//     PlcTask Inputs/GVL_iXlinker.EtherCAT_Master_EMxxxx.Beckhoff_EM7xxx.A_0006_EM7004_0000_0018.ENC_Inputs_Channel_3.Latch_value <-> ENC Inputs Channel 3/Latch value
//     PlcTask Inputs/GVL_iXlinker.EtherCAT_Master_EMxxxx.Beckhoff_EM7xxx.A_0006_EM7004_0000_0018.ENC_Inputs_Channel_4.Latch_value <-> ENC Inputs Channel 4/Latch value
//     PlcTask Inputs/GVL_iXlinker.EtherCAT_Master_EMxxxx.Beckhoff_EM7xxx.A_0006_EM7004_0000_0018.PLS_Inputs.Status/PLS_Enabled <-> PLS Inputs/Status/PLS Enabled
//     PlcTask Inputs/GVL_iXlinker.EtherCAT_Master_EMxxxx.Beckhoff_EM7xxx.A_0006_EM7004_0000_0018.PLS_Inputs.Status/Unequal_SI_0 <-> PLS Inputs/Status/Unequal SI:0
//     PlcTask Outputs/GVL_iXlinker.EtherCAT_Master_EMxxxx.Beckhoff_EM7xxx.A_0006_EM7004_0000_0018.DO_Outputs.Output/Output_0 <-> DO Outputs/Output/Output 0
//     PlcTask Outputs/GVL_iXlinker.EtherCAT_Master_EMxxxx.Beckhoff_EM7xxx.A_0006_EM7004_0000_0018.DO_Outputs.Output/Output_1 <-> DO Outputs/Output/Output 1
//     PlcTask Outputs/GVL_iXlinker.EtherCAT_Master_EMxxxx.Beckhoff_EM7xxx.A_0006_EM7004_0000_0018.DO_Outputs.Output/Output_2 <-> DO Outputs/Output/Output 2
//     PlcTask Outputs/GVL_iXlinker.EtherCAT_Master_EMxxxx.Beckhoff_EM7xxx.A_0006_EM7004_0000_0018.DO_Outputs.Output/Output_3 <-> DO Outputs/Output/Output 3
//     PlcTask Outputs/GVL_iXlinker.EtherCAT_Master_EMxxxx.Beckhoff_EM7xxx.A_0006_EM7004_0000_0018.DO_Outputs.Output/Output_4 <-> DO Outputs/Output/Output 4
//     PlcTask Outputs/GVL_iXlinker.EtherCAT_Master_EMxxxx.Beckhoff_EM7xxx.A_0006_EM7004_0000_0018.DO_Outputs.Output/Output_5 <-> DO Outputs/Output/Output 5
//     PlcTask Outputs/GVL_iXlinker.EtherCAT_Master_EMxxxx.Beckhoff_EM7xxx.A_0006_EM7004_0000_0018.DO_Outputs.Output/Output_6 <-> DO Outputs/Output/Output 6
//     PlcTask Outputs/GVL_iXlinker.EtherCAT_Master_EMxxxx.Beckhoff_EM7xxx.A_0006_EM7004_0000_0018.DO_Outputs.Output/Output_7 <-> DO Outputs/Output/Output 7
//     PlcTask Outputs/GVL_iXlinker.EtherCAT_Master_EMxxxx.Beckhoff_EM7xxx.A_0006_EM7004_0000_0018.DO_Outputs.Output/Output_8 <-> DO Outputs/Output/Output 8
//     PlcTask Outputs/GVL_iXlinker.EtherCAT_Master_EMxxxx.Beckhoff_EM7xxx.A_0006_EM7004_0000_0018.DO_Outputs.Output/Output_9 <-> DO Outputs/Output/Output 9
//     PlcTask Outputs/GVL_iXlinker.EtherCAT_Master_EMxxxx.Beckhoff_EM7xxx.A_0006_EM7004_0000_0018.DO_Outputs.Output/Output_10 <-> DO Outputs/Output/Output 10
//     PlcTask Outputs/GVL_iXlinker.EtherCAT_Master_EMxxxx.Beckhoff_EM7xxx.A_0006_EM7004_0000_0018.DO_Outputs.Output/Output_11 <-> DO Outputs/Output/Output 11
//     PlcTask Outputs/GVL_iXlinker.EtherCAT_Master_EMxxxx.Beckhoff_EM7xxx.A_0006_EM7004_0000_0018.DO_Outputs.Output/Output_12 <-> DO Outputs/Output/Output 12
//     PlcTask Outputs/GVL_iXlinker.EtherCAT_Master_EMxxxx.Beckhoff_EM7xxx.A_0006_EM7004_0000_0018.DO_Outputs.Output/Output_13 <-> DO Outputs/Output/Output 13
//     PlcTask Outputs/GVL_iXlinker.EtherCAT_Master_EMxxxx.Beckhoff_EM7xxx.A_0006_EM7004_0000_0018.DO_Outputs.Output/Output_14 <-> DO Outputs/Output/Output 14
//     PlcTask Outputs/GVL_iXlinker.EtherCAT_Master_EMxxxx.Beckhoff_EM7xxx.A_0006_EM7004_0000_0018.DO_Outputs.Output/Output_15 <-> DO Outputs/Output/Output 15
//     PlcTask Outputs/GVL_iXlinker.EtherCAT_Master_EMxxxx.Beckhoff_EM7xxx.A_0006_EM7004_0000_0018.AO_Outputs_Channel_1.Analog_output <-> AO Outputs Channel 1/Analog output
//     PlcTask Outputs/GVL_iXlinker.EtherCAT_Master_EMxxxx.Beckhoff_EM7xxx.A_0006_EM7004_0000_0018.AO_Outputs_Channel_2.Analog_output <-> AO Outputs Channel 2/Analog output
//     PlcTask Outputs/GVL_iXlinker.EtherCAT_Master_EMxxxx.Beckhoff_EM7xxx.A_0006_EM7004_0000_0018.AO_Outputs_Channel_3.Analog_output <-> AO Outputs Channel 3/Analog output
//     PlcTask Outputs/GVL_iXlinker.EtherCAT_Master_EMxxxx.Beckhoff_EM7xxx.A_0006_EM7004_0000_0018.AO_Outputs_Channel_4.Analog_output <-> AO Outputs Channel 4/Analog output
//     PlcTask Outputs/GVL_iXlinker.EtherCAT_Master_EMxxxx.Beckhoff_EM7xxx.A_0006_EM7004_0000_0018.ENC_Outputs_Channel_1.Control/Enable_latch_extern_on_positive_edge <-> ENC Outputs Channel 1/Control/Enable latch extern on positive edge
//     PlcTask Outputs/GVL_iXlinker.EtherCAT_Master_EMxxxx.Beckhoff_EM7xxx.A_0006_EM7004_0000_0018.ENC_Outputs_Channel_2.Control/Enable_latch_extern_on_positive_edge <-> ENC Outputs Channel 2/Control/Enable latch extern on positive edge
//     PlcTask Outputs/GVL_iXlinker.EtherCAT_Master_EMxxxx.Beckhoff_EM7xxx.A_0006_EM7004_0000_0018.ENC_Outputs_Channel_3.Control/Enable_latch_extern_on_positive_edge <-> ENC Outputs Channel 3/Control/Enable latch extern on positive edge
//     PlcTask Outputs/GVL_iXlinker.EtherCAT_Master_EMxxxx.Beckhoff_EM7xxx.A_0006_EM7004_0000_0018.ENC_Outputs_Channel_4.Control/Enable_latch_extern_on_positive_edge <-> ENC Outputs Channel 4/Control/Enable latch extern on positive edge
//     PlcTask Outputs/GVL_iXlinker.EtherCAT_Master_EMxxxx.Beckhoff_EM7xxx.A_0006_EM7004_0000_0018.ENC_Outputs_Channel_1.Control/Set_counter <-> ENC Outputs Channel 1/Control/Set counter
//     PlcTask Outputs/GVL_iXlinker.EtherCAT_Master_EMxxxx.Beckhoff_EM7xxx.A_0006_EM7004_0000_0018.ENC_Outputs_Channel_2.Control/Set_counter <-> ENC Outputs Channel 2/Control/Set counter
//     PlcTask Outputs/GVL_iXlinker.EtherCAT_Master_EMxxxx.Beckhoff_EM7xxx.A_0006_EM7004_0000_0018.ENC_Outputs_Channel_3.Control/Set_counter <-> ENC Outputs Channel 3/Control/Set counter
//     PlcTask Outputs/GVL_iXlinker.EtherCAT_Master_EMxxxx.Beckhoff_EM7xxx.A_0006_EM7004_0000_0018.ENC_Outputs_Channel_4.Control/Set_counter <-> ENC Outputs Channel 4/Control/Set counter
//     PlcTask Outputs/GVL_iXlinker.EtherCAT_Master_EMxxxx.Beckhoff_EM7xxx.A_0006_EM7004_0000_0018.ENC_Outputs_Channel_1.Control/Enable_latch_extern_on_negative_edge <-> ENC Outputs Channel 1/Control/Enable latch extern on negative edge
//     PlcTask Outputs/GVL_iXlinker.EtherCAT_Master_EMxxxx.Beckhoff_EM7xxx.A_0006_EM7004_0000_0018.ENC_Outputs_Channel_2.Control/Enable_latch_extern_on_negative_edge <-> ENC Outputs Channel 2/Control/Enable latch extern on negative edge
//     PlcTask Outputs/GVL_iXlinker.EtherCAT_Master_EMxxxx.Beckhoff_EM7xxx.A_0006_EM7004_0000_0018.ENC_Outputs_Channel_3.Control/Enable_latch_extern_on_negative_edge <-> ENC Outputs Channel 3/Control/Enable latch extern on negative edge
//     PlcTask Outputs/GVL_iXlinker.EtherCAT_Master_EMxxxx.Beckhoff_EM7xxx.A_0006_EM7004_0000_0018.ENC_Outputs_Channel_4.Control/Enable_latch_extern_on_negative_edge <-> ENC Outputs Channel 4/Control/Enable latch extern on negative edge
//     PlcTask Outputs/GVL_iXlinker.EtherCAT_Master_EMxxxx.Beckhoff_EM7xxx.A_0006_EM7004_0000_0018.ENC_Outputs_Channel_1.Set_counter_value <-> ENC Outputs Channel 1/Set counter value
//     PlcTask Outputs/GVL_iXlinker.EtherCAT_Master_EMxxxx.Beckhoff_EM7xxx.A_0006_EM7004_0000_0018.ENC_Outputs_Channel_2.Set_counter_value <-> ENC Outputs Channel 2/Set counter value
//     PlcTask Outputs/GVL_iXlinker.EtherCAT_Master_EMxxxx.Beckhoff_EM7xxx.A_0006_EM7004_0000_0018.ENC_Outputs_Channel_3.Set_counter_value <-> ENC Outputs Channel 3/Set counter value
//     PlcTask Outputs/GVL_iXlinker.EtherCAT_Master_EMxxxx.Beckhoff_EM7xxx.A_0006_EM7004_0000_0018.ENC_Outputs_Channel_4.Set_counter_value <-> ENC Outputs Channel 4/Set counter value
//     PlcTask Outputs/GVL_iXlinker.EtherCAT_Master_EMxxxx.Beckhoff_EM7xxx.A_0006_EM7004_0000_0018.PLS_Outputs.Control/Enable_PLS <-> PLS Outputs/Control/Enable PLS
//     PlcTask Inputs/GVL_iXlinker.EtherCAT_Master_EMxxxx.Beckhoff_EM7xxx.A_0006_EM7004_0000_0018.WcState.WcState <-> WcState/WcState
//     PlcTask Inputs/GVL_iXlinker.EtherCAT_Master_EMxxxx.Beckhoff_EM7xxx.A_0006_EM7004_0000_0018.WcState.InputToggle <-> WcState/InputToggle
//     PlcTask Inputs/GVL_iXlinker.EtherCAT_Master_EMxxxx.Beckhoff_EM7xxx.A_0006_EM7004_0000_0018.InfoData.AdsAddr <-> InfoData/AdsAddr
//     PlcTask Inputs/GVL_iXlinker.EtherCAT_Master_EMxxxx.Beckhoff_EM7xxx.A_0006_EM7004_0000_0018.InfoData.State <-> InfoData/State
//   PLC/PLC Instance <-> EtherCAT_Master_EMxxxx
//     PlcTask Inputs/GVL_iXlinker.EtherCAT_Master_EMxxxx.SyncUnits._default._unreferenced.WcState.WcState <-> SyncUnits/<default>/<unreferenced>/WcState/WcState
//     PlcTask Inputs/GVL_iXlinker.EtherCAT_Master_EMxxxx.SyncUnits._default._unreferenced.InfoData.ObjectId <-> SyncUnits/<default>/<unreferenced>/InfoData/ObjectId
//     PlcTask Inputs/GVL_iXlinker.EtherCAT_Master_EMxxxx.SyncUnits._default._unreferenced.InfoData.State <-> SyncUnits/<default>/<unreferenced>/InfoData/State
//     PlcTask Inputs/GVL_iXlinker.EtherCAT_Master_EMxxxx.SyncUnits._default._unreferenced.InfoData.SlaveCount <-> SyncUnits/<default>/<unreferenced>/InfoData/SlaveCount
//     PlcTask Inputs/GVL_iXlinker.EtherCAT_Master_EMxxxx.SyncUnits._default.PlcTask.WcState.WcState <-> SyncUnits/<default>/PlcTask/WcState/WcState
//     PlcTask Inputs/GVL_iXlinker.EtherCAT_Master_EMxxxx.SyncUnits._default.PlcTask.InfoData.ObjectId <-> SyncUnits/<default>/PlcTask/InfoData/ObjectId
//     PlcTask Inputs/GVL_iXlinker.EtherCAT_Master_EMxxxx.SyncUnits._default.PlcTask.InfoData.State <-> SyncUnits/<default>/PlcTask/InfoData/State
//     PlcTask Inputs/GVL_iXlinker.EtherCAT_Master_EMxxxx.SyncUnits._default.PlcTask.InfoData.SlaveCount <-> SyncUnits/<default>/PlcTask/InfoData/SlaveCount
//     PlcTask Inputs/GVL_iXlinker.EtherCAT_Master_EMxxxx.Inputs.SlaveCount <-> Inputs/SlaveCount
//     PlcTask Inputs/GVL_iXlinker.EtherCAT_Master_EMxxxx.Inputs.DevState <-> Inputs/DevState
//     PlcTask Inputs/GVL_iXlinker.EtherCAT_Master_EMxxxx.Inputs.Frm{0..25}State <-> Inputs/Frm{0..25}State  (26 links)
//     PlcTask Inputs/GVL_iXlinker.EtherCAT_Master_EMxxxx.Inputs.Frm{0..25}WcState <-> Inputs/Frm{0..25}WcState  (26 links)
//     PlcTask Inputs/GVL_iXlinker.EtherCAT_Master_EMxxxx.Inputs.Frm{0..25}InputToggle <-> Inputs/Frm{0..25}InputToggle  (26 links)
//     PlcTask Outputs/GVL_iXlinker.EtherCAT_Master_EMxxxx.Outputs.DevCtrl <-> Outputs/DevCtrl
//     PlcTask Outputs/GVL_iXlinker.EtherCAT_Master_EMxxxx.Outputs.Frm{0..25}Ctrl <-> Outputs/Frm{0..25}Ctrl  (26 links)
//     PlcTask Outputs/GVL_iXlinker.EtherCAT_Master_EMxxxx.Outputs.Frm{0..25}WcCtrl <-> Outputs/Frm{0..25}WcCtrl  (26 links)
//     PlcTask Inputs/GVL_iXlinker.EtherCAT_Master_EMxxxx.InfoData.ChangeCount <-> InfoData/ChangeCount
//     PlcTask Inputs/GVL_iXlinker.EtherCAT_Master_EMxxxx.InfoData.DevId <-> InfoData/DevId
//     PlcTask Inputs/GVL_iXlinker.EtherCAT_Master_EMxxxx.InfoData.AmsNetId <-> InfoData/AmsNetId
//     PlcTask Inputs/GVL_iXlinker.EtherCAT_Master_EMxxxx.InfoData.CfgSlaveCount <-> InfoData/CfgSlaveCount
//     PlcTask Inputs/GVL_iXlinker.EtherCAT_Master_EMxxxx.InfoData.DcToTcTimeOffset <-> InfoData/DcToTcTimeOffset
//     PlcTask Inputs/GVL_iXlinker.EtherCAT_Master_EMxxxx.InfoData.DcToExtTimeOffset <-> InfoData/DcToExtTimeOffset

CONFIGURATION PLC
    RESOURCE PLC ON TwinCAT3
        TASK PlcTask(INTERVAL := T#10ms, PRIORITY := 20);
        PROGRAM MAIN WITH PlcTask : MAIN;
    END_RESOURCE
END_CONFIGURATION

// ---- DUTs/IO/PdoEntries/Status_E3F6A94B.TcDUT
{attribute 'GeneratedUsingTerminal: EM3701-0000-0016'}
{attribute addProperty BoxType "EM3701-0000-0016"}
{attribute addProperty Id "UnderrangeBOOL1OverrangeBOOL1Limit_1BYTE1Limit_2BYTE1ErrorBOOL1TxPDO_StateBOOL1"}
{attribute addProperty CRC "3824593227"}
{attribute addProperty Size "6"}
TYPE Status_E3F6A94B :
STRUCT
	{attribute addProperty Name "Underrange"}
	Underrange : BOOL;
	{attribute addProperty Name "Overrange"}
	Overrange : BOOL;
	{attribute addProperty Name "Limit_1"}
	Limit_1 : BYTE;
	{attribute addProperty Name "Limit_2"}
	Limit_2 : BYTE;
	{attribute addProperty Name "Error"}
	Error : BOOL;
	{attribute addProperty Name "TxPDO_State"}
	TxPDO_State : BOOL;
END_STRUCT
END_TYPE

// ---- DUTs/IO/PdoEntries/Input_97D1F313.TcDUT
{attribute 'GeneratedUsingTerminal: EM7004-0000-0017'}
{attribute addProperty BoxType "EM7004-0000-0017"}
{attribute addProperty Id "Input_0BOOL1Input_1BOOL1Input_2BOOL1Input_3BOOL1Input_4BOOL1Input_5BOOL1Input_6BOOL1Input_7BOOL1Input_8BOOL1Input_9BOOL1Input_10BOOL1Input_11BOOL1Input_12BOOL1Input_13BOOL1Input_14BOOL1Input_15BOOL1"}
{attribute addProperty CRC "2547118867"}
{attribute addProperty Size "16"}
TYPE Input_97D1F313 :
STRUCT
	{attribute addProperty Name "Input_0"}
	Input_0 : BOOL;
	{attribute addProperty Name "Input_1"}
	Input_1 : BOOL;
	{attribute addProperty Name "Input_2"}
	Input_2 : BOOL;
	{attribute addProperty Name "Input_3"}
	Input_3 : BOOL;
	{attribute addProperty Name "Input_4"}
	Input_4 : BOOL;
	{attribute addProperty Name "Input_5"}
	Input_5 : BOOL;
	{attribute addProperty Name "Input_6"}
	Input_6 : BOOL;
	{attribute addProperty Name "Input_7"}
	Input_7 : BOOL;
	{attribute addProperty Name "Input_8"}
	Input_8 : BOOL;
	{attribute addProperty Name "Input_9"}
	Input_9 : BOOL;
	{attribute addProperty Name "Input_10"}
	Input_10 : BOOL;
	{attribute addProperty Name "Input_11"}
	Input_11 : BOOL;
	{attribute addProperty Name "Input_12"}
	Input_12 : BOOL;
	{attribute addProperty Name "Input_13"}
	Input_13 : BOOL;
	{attribute addProperty Name "Input_14"}
	Input_14 : BOOL;
	{attribute addProperty Name "Input_15"}
	Input_15 : BOOL;
END_STRUCT
END_TYPE

// ---- DUTs/IO/PdoEntries/Status_B4798D86.TcDUT
{attribute 'GeneratedUsingTerminal: EM7004-0000-0017'}
{attribute addProperty BoxType "EM7004-0000-0017"}
{attribute addProperty Id "Latch_extern_validBOOL1Set_counter_doneBOOL1Status_of_input_ABOOL1Status_of_input_BBOOL1Status_of_input_gateBOOL1Status_of_extern_latchBOOL1TxPDO_ToggleBOOL1"}
{attribute addProperty CRC "3027864966"}
{attribute addProperty Size "7"}
TYPE Status_B4798D86 :
STRUCT
	{attribute addProperty Name "Latch_extern_valid"}
	Latch_extern_valid : BOOL;
	{attribute addProperty Name "Set_counter_done"}
	Set_counter_done : BOOL;
	{attribute addProperty Name "Status_of_input_A"}
	Status_of_input_A : BOOL;
	{attribute addProperty Name "Status_of_input_B"}
	Status_of_input_B : BOOL;
	{attribute addProperty Name "Status_of_input_gate"}
	Status_of_input_gate : BOOL;
	{attribute addProperty Name "Status_of_extern_latch"}
	Status_of_extern_latch : BOOL;
	{attribute addProperty Name "TxPDO_Toggle"}
	TxPDO_Toggle : BOOL;
END_STRUCT
END_TYPE

// ---- DUTs/IO/PdoEntries/Status_882A150F.TcDUT
{attribute 'GeneratedUsingTerminal: EM7004-0000-0017'}
{attribute addProperty BoxType "EM7004-0000-0017"}
{attribute addProperty Id "PLS_EnabledBOOL1Unequal_SI_0BOOL1"}
{attribute addProperty CRC "2284459279"}
{attribute addProperty Size "2"}
TYPE Status_882A150F :
STRUCT
	{attribute addProperty Name "PLS_Enabled"}
	PLS_Enabled : BOOL;
	{attribute addProperty Name "Unequal_SI_0"}
	Unequal_SI_0 : BOOL;
END_STRUCT
END_TYPE

// ---- DUTs/IO/PdoEntries/Output_FFFF807A.TcDUT
{attribute 'GeneratedUsingTerminal: EM7004-0000-0017'}
{attribute addProperty BoxType "EM7004-0000-0017"}
{attribute addProperty Id "Output_0BOOL1Output_1BOOL1Output_2BOOL1Output_3BOOL1Output_4BOOL1Output_5BOOL1Output_6BOOL1Output_7BOOL1Output_8BOOL1Output_9BOOL1Output_10BOOL1Output_11BOOL1Output_12BOOL1Output_13BOOL1Output_14BOOL1Output_15BOOL1"}
{attribute addProperty CRC "4294934650"}
{attribute addProperty Size "16"}
TYPE Output_FFFF807A :
STRUCT
	{attribute addProperty Name "Output_0"}
	Output_0 : BOOL;
	{attribute addProperty Name "Output_1"}
	Output_1 : BOOL;
	{attribute addProperty Name "Output_2"}
	Output_2 : BOOL;
	{attribute addProperty Name "Output_3"}
	Output_3 : BOOL;
	{attribute addProperty Name "Output_4"}
	Output_4 : BOOL;
	{attribute addProperty Name "Output_5"}
	Output_5 : BOOL;
	{attribute addProperty Name "Output_6"}
	Output_6 : BOOL;
	{attribute addProperty Name "Output_7"}
	Output_7 : BOOL;
	{attribute addProperty Name "Output_8"}
	Output_8 : BOOL;
	{attribute addProperty Name "Output_9"}
	Output_9 : BOOL;
	{attribute addProperty Name "Output_10"}
	Output_10 : BOOL;
	{attribute addProperty Name "Output_11"}
	Output_11 : BOOL;
	{attribute addProperty Name "Output_12"}
	Output_12 : BOOL;
	{attribute addProperty Name "Output_13"}
	Output_13 : BOOL;
	{attribute addProperty Name "Output_14"}
	Output_14 : BOOL;
	{attribute addProperty Name "Output_15"}
	Output_15 : BOOL;
END_STRUCT
END_TYPE

// ---- DUTs/IO/PdoEntries/Control_F189B737.TcDUT
{attribute 'GeneratedUsingTerminal: EM7004-0000-0017'}
{attribute addProperty BoxType "EM7004-0000-0017"}
{attribute addProperty Id "Enable_latch_extern_on_positive_edgeBOOL1Set_counterBOOL1Enable_latch_extern_on_negative_edgeBOOL1"}
{attribute addProperty CRC "4052334391"}
{attribute addProperty Size "3"}
TYPE Control_F189B737 :
STRUCT
	{attribute addProperty Name "Enable_latch_extern_on_positive_edge"}
	Enable_latch_extern_on_positive_edge : BOOL;
	{attribute addProperty Name "Set_counter"}
	Set_counter : BOOL;
	{attribute addProperty Name "Enable_latch_extern_on_negative_edge"}
	Enable_latch_extern_on_negative_edge : BOOL;
END_STRUCT
END_TYPE

// ---- DUTs/IO/PdoEntries/Control_17BA1FC2.TcDUT
{attribute 'GeneratedUsingTerminal: EM7004-0000-0017'}
{attribute addProperty BoxType "EM7004-0000-0017"}
{attribute addProperty Id "Enable_PLSBOOL1"}
{attribute addProperty CRC "398073794"}
{attribute addProperty Size "1"}
TYPE Control_17BA1FC2 :
STRUCT
	{attribute addProperty Name "Enable_PLS"}
	Enable_PLS : BOOL;
END_STRUCT
END_TYPE

// ---- DUTs/IO/PDOs/InfoData_6F19DB2B.TcDUT
{attribute 'GeneratedUsingTerminal: EK1100-0000-0018'}
{attribute addProperty BoxType "EK1100-0000-0018"}
{attribute addProperty Id "StateAT %I*UINT2"}
{attribute addProperty CRC "1863965483"}
{attribute addProperty Size "2"}
TYPE InfoData_6F19DB2B :
STRUCT
	{attribute addProperty Name "State"}
	State AT %I* : UINT;
END_STRUCT
END_TYPE

// ---- DUTs/IO/PDOs/Channel_42CA91F7.TcDUT
{attribute 'GeneratedUsingTerminal: EM2042-0000-0016'}
{attribute addProperty BoxType "EM2042-0000-0016"}
{attribute addProperty Id "OutputAT %Q*BOOL1"}
{attribute addProperty CRC "1120571895"}
{attribute addProperty Size "1"}
TYPE Channel_42CA91F7 EXTENDS OutputBase_10CEE7DE :
STRUCT
	{attribute addProperty Name "Output"}
	Output AT %Q* : BOOL;
END_STRUCT
END_TYPE

// ---- DUTs/IO/PDOs/WcState_0B2B16F9.TcDUT
{attribute 'GeneratedUsingTerminal: EM2042-0000-0016'}
{attribute addProperty BoxType "EM2042-0000-0016"}
{attribute addProperty Id "WcStateAT %I*BOOL1"}
{attribute addProperty CRC "187373305"}
{attribute addProperty Size "1"}
TYPE WcState_0B2B16F9 :
STRUCT
	{attribute addProperty Name "WcState"}
	WcState AT %I* : BOOL;
END_STRUCT
END_TYPE

// ---- DUTs/IO/PDOs/AI_Inputs_5AF6604E.TcDUT
{attribute 'GeneratedUsingTerminal: EM3701-0000-0016'}
{attribute addProperty BoxType "EM3701-0000-0016"}
{attribute addProperty Id "StatusAT %I*Status_E3F6A94B6ValueAT %I*INT2"}
{attribute addProperty CRC "1526095950"}
{attribute addProperty Size "8"}
TYPE AI_Inputs_5AF6604E EXTENDS InputBase_8311D824 :
STRUCT
	{attribute addProperty Name "Status"}
	Status AT %I* : Status_E3F6A94B;
	{attribute addProperty Name "Value"}
	Value AT %I* : INT;
END_STRUCT
END_TYPE

// ---- DUTs/IO/PDOs/WcState_9091E0EB.TcDUT
{attribute 'GeneratedUsingTerminal: EM3701-0000-0016'}
{attribute addProperty BoxType "EM3701-0000-0016"}
{attribute addProperty Id "WcStateAT %I*BOOL1InputToggleAT %I*BOOL1"}
{attribute addProperty CRC "2425479403"}
{attribute addProperty Size "2"}
TYPE WcState_9091E0EB :
STRUCT
	{attribute addProperty Name "WcState"}
	WcState AT %I* : BOOL;
	{attribute addProperty Name "InputToggle"}
	InputToggle AT %I* : BOOL;
END_STRUCT
END_TYPE

// ---- DUTs/IO/PDOs/InfoData_32EB74EA.TcDUT
{attribute 'GeneratedUsingTerminal: EM3701-0000-0016'}
{attribute addProperty BoxType "EM3701-0000-0016"}
{attribute addProperty Id "AdsAddrAT %I*AMSADDR8StateAT %I*UINT2"}
{attribute addProperty CRC "854291690"}
{attribute addProperty Size "10"}
TYPE InfoData_32EB74EA EXTENDS InputBase_8311D824 :
STRUCT
	{attribute addProperty Name "AdsAddr"}
	AdsAddr AT %I* : AMSADDR;
	{attribute addProperty Name "State"}
	State AT %I* : UINT;
END_STRUCT
END_TYPE

// ---- DUTs/IO/PDOs/AI_Input_Channel_5AF6604E.TcDUT
{attribute 'GeneratedUsingTerminal: EM3702-0000-0016'}
{attribute addProperty BoxType "EM3702-0000-0016"}
{attribute addProperty Id "StatusAT %I*Status_E3F6A94B6ValueAT %I*INT2"}
{attribute addProperty CRC "1526095950"}
{attribute addProperty Size "8"}
TYPE AI_Input_Channel_5AF6604E EXTENDS InputBase_8311D824 :
STRUCT
	{attribute addProperty Name "Status"}
	Status AT %I* : Status_E3F6A94B;
	{attribute addProperty Name "Value"}
	Value AT %I* : INT;
END_STRUCT
END_TYPE

// ---- DUTs/IO/PDOs/Digital_BD004D6F.TcDUT
{attribute 'GeneratedUsingTerminal: EM7004-0000-9995'}
{attribute addProperty BoxType "EM7004-0000-9995"}
{attribute addProperty Id "InputAT %I*ARRAY[0..15] OF BOOL16"}
{attribute addProperty CRC "2621435360"}
{attribute addProperty Size "16"}
TYPE Digital_BD004D6F EXTENDS InputBase_8311D824 :
STRUCT
	{attribute addProperty Name "Input"}
	Input AT %I* : ARRAY[0..15] OF BOOL;
END_STRUCT
END_TYPE

// ---- DUTs/IO/PDOs/Encoder_Channel_2E4EA213.TcDUT
{attribute 'GeneratedUsingTerminal: EM7004-0000-9995'}
{attribute addProperty BoxType "EM7004-0000-9995"}
{attribute addProperty Id "StatusAT %I*UINT2ValueAT %I*UINT2LatchAT %I*UINT2"}
{attribute addProperty CRC "776905235"}
{attribute addProperty Size "6"}
TYPE Encoder_Channel_2E4EA213 EXTENDS InputBase_8311D824 :
STRUCT
	{attribute addProperty Name "Status"}
	Status AT %I* : UINT;
	{attribute addProperty Name "Value"}
	Value AT %I* : UINT;
	{attribute addProperty Name "Latch"}
	Latch AT %I* : UINT;
END_STRUCT
END_TYPE

// ---- DUTs/IO/PDOs/Digital_A7E1DFAB.TcDUT
{attribute 'GeneratedUsingTerminal: EM7004-0000-9995'}
{attribute addProperty BoxType "EM7004-0000-9995"}
{attribute addProperty Id "OutputAT %Q*ARRAY[0..15] OF BOOL16"}
{attribute addProperty CRC "1538723034"}
{attribute addProperty Size "16"}
TYPE Digital_A7E1DFAB EXTENDS OutputBase_10CEE7DE :
STRUCT
	{attribute addProperty Name "Output"}
	Output AT %Q* : ARRAY[0..15] OF BOOL;
END_STRUCT
END_TYPE

// ---- DUTs/IO/PDOs/Analog_Channel_5F9B7EA6.TcDUT
{attribute 'GeneratedUsingTerminal: EM7004-0000-9995'}
{attribute addProperty BoxType "EM7004-0000-9995"}
{attribute addProperty Id "OutputAT %Q*INT2"}
{attribute addProperty CRC "1604026022"}
{attribute addProperty Size "2"}
TYPE Analog_Channel_5F9B7EA6 EXTENDS OutputBase_10CEE7DE :
STRUCT
	{attribute addProperty Name "Output"}
	Output AT %Q* : INT;
END_STRUCT
END_TYPE

// ---- DUTs/IO/PDOs/Encoder_Channel_B7999E14.TcDUT
{attribute 'GeneratedUsingTerminal: EM7004-0000-9995'}
{attribute addProperty BoxType "EM7004-0000-9995"}
{attribute addProperty Id "CtrlAT %Q*UINT2ValueAT %Q*UINT2"}
{attribute addProperty CRC "3080298004"}
{attribute addProperty Size "4"}
TYPE Encoder_Channel_B7999E14 EXTENDS OutputBase_10CEE7DE :
STRUCT
	{attribute addProperty Name "Ctrl"}
	Ctrl AT %Q* : UINT;
	{attribute addProperty Name "Value"}
	Value AT %Q* : UINT;
END_STRUCT
END_TYPE

// ---- DUTs/IO/PDOs/DI_Inputs_BD004D6F.TcDUT
{attribute 'GeneratedUsingTerminal: EM7004-0000-9996'}
{attribute addProperty BoxType "EM7004-0000-9996"}
{attribute addProperty Id "InputAT %I*ARRAY[0..15] OF BOOL16"}
{attribute addProperty CRC "2621435360"}
{attribute addProperty Size "16"}
TYPE DI_Inputs_BD004D6F EXTENDS InputBase_8311D824 :
STRUCT
	{attribute addProperty Name "Input"}
	Input AT %I* : ARRAY[0..15] OF BOOL;
END_STRUCT
END_TYPE

// ---- DUTs/IO/PDOs/ENC_Inputs_Channel_69C51E8E.TcDUT
{attribute 'GeneratedUsingTerminal: EM7004-0000-9996'}
{attribute addProperty BoxType "EM7004-0000-9996"}
{attribute addProperty Id "Latch_extern_validAT %I*BOOL1Set_counter_doneAT %I*BOOL1Status_of_input_AAT %I*BOOL1Status_of_input_BAT %I*BOOL1Status_of_input_gateAT %I*BOOL1Status_of_extern_latchAT %I*BOOL1Counter_valueAT %I*UINT2Latch_valueAT %I*UINT2"}
{attribute addProperty CRC "1774526094"}
{attribute addProperty Size "10"}
TYPE ENC_Inputs_Channel_69C51E8E EXTENDS InputBase_8311D824 :
STRUCT
	{attribute addProperty Name "Latch_extern_valid"}
	Latch_extern_valid AT %I* : BOOL;
	{attribute addProperty Name "Set_counter_done"}
	Set_counter_done AT %I* : BOOL;
	{attribute addProperty Name "Status_of_input_A"}
	Status_of_input_A AT %I* : BOOL;
	{attribute addProperty Name "Status_of_input_B"}
	Status_of_input_B AT %I* : BOOL;
	{attribute addProperty Name "Status_of_input_gate"}
	Status_of_input_gate AT %I* : BOOL;
	{attribute addProperty Name "Status_of_extern_latch"}
	Status_of_extern_latch AT %I* : BOOL;
	{attribute addProperty Name "Counter_value"}
	Counter_value AT %I* : UINT;
	{attribute addProperty Name "Latch_value"}
	Latch_value AT %I* : UINT;
END_STRUCT
END_TYPE

// ---- DUTs/IO/PDOs/PLS_Inputs_5A35B63D.TcDUT
{attribute 'GeneratedUsingTerminal: EM7004-0000-9996'}
{attribute addProperty BoxType "EM7004-0000-9996"}
{attribute addProperty Id "PLS_EnabledAT %I*BOOL1Unequal_SI_0AT %I*BOOL1"}
{attribute addProperty CRC "1513469501"}
{attribute addProperty Size "2"}
TYPE PLS_Inputs_5A35B63D EXTENDS InputBase_8311D824 :
STRUCT
	{attribute addProperty Name "PLS_Enabled"}
	PLS_Enabled AT %I* : BOOL;
	{attribute addProperty Name "Unequal_SI_0"}
	Unequal_SI_0 AT %I* : BOOL;
END_STRUCT
END_TYPE

// ---- DUTs/IO/PDOs/DO_Outputs_A7E1DFAB.TcDUT
{attribute 'GeneratedUsingTerminal: EM7004-0000-9996'}
{attribute addProperty BoxType "EM7004-0000-9996"}
{attribute addProperty Id "OutputAT %Q*ARRAY[0..15] OF BOOL16"}
{attribute addProperty CRC "1538723034"}
{attribute addProperty Size "16"}
TYPE DO_Outputs_A7E1DFAB EXTENDS OutputBase_10CEE7DE :
STRUCT
	{attribute addProperty Name "Output"}
	Output AT %Q* : ARRAY[0..15] OF BOOL;
END_STRUCT
END_TYPE

// ---- DUTs/IO/PDOs/AO_Output_Channel_BA7EBB7C.TcDUT
{attribute 'GeneratedUsingTerminal: EM7004-0000-9996'}
{attribute addProperty BoxType "EM7004-0000-9996"}
{attribute addProperty Id "Analog_outputAT %Q*INT2"}
{attribute addProperty CRC "3128867708"}
{attribute addProperty Size "2"}
TYPE AO_Output_Channel_BA7EBB7C EXTENDS OutputBase_10CEE7DE :
STRUCT
	{attribute addProperty Name "Analog_output"}
	Analog_output AT %Q* : INT;
END_STRUCT
END_TYPE

// ---- DUTs/IO/PDOs/ENC_Outputs_Channel_DC4E290B.TcDUT
{attribute 'GeneratedUsingTerminal: EM7004-0000-9996'}
{attribute addProperty BoxType "EM7004-0000-9996"}
{attribute addProperty Id "Enable_latch_extern_on_positive_edgeAT %Q*BOOL1Set_counterAT %Q*BOOL1Enable_latch_extern_on_negative_edgeAT %Q*BOOL1Set_counter_valueAT %Q*UINT2"}
{attribute addProperty CRC "3696109835"}
{attribute addProperty Size "5"}
TYPE ENC_Outputs_Channel_DC4E290B EXTENDS OutputBase_10CEE7DE :
STRUCT
	{attribute addProperty Name "Enable_latch_extern_on_positive_edge"}
	Enable_latch_extern_on_positive_edge AT %Q* : BOOL;
	{attribute addProperty Name "Set_counter"}
	Set_counter AT %Q* : BOOL;
	{attribute addProperty Name "Enable_latch_extern_on_negative_edge"}
	Enable_latch_extern_on_negative_edge AT %Q* : BOOL;
	{attribute addProperty Name "Set_counter_value"}
	Set_counter_value AT %Q* : UINT;
END_STRUCT
END_TYPE

// ---- DUTs/IO/PDOs/PLS_Outputs_AFB7DAF5.TcDUT
{attribute 'GeneratedUsingTerminal: EM7004-0000-9996'}
{attribute addProperty BoxType "EM7004-0000-9996"}
{attribute addProperty Id "Enable_PLSAT %Q*BOOL1"}
{attribute addProperty CRC "2948061941"}
{attribute addProperty Size "1"}
TYPE PLS_Outputs_AFB7DAF5 EXTENDS OutputBase_10CEE7DE :
STRUCT
	{attribute addProperty Name "Enable_PLS"}
	Enable_PLS AT %Q* : BOOL;
END_STRUCT
END_TYPE

// ---- DUTs/IO/PDOs/ENC_Inputs_Channel_6B6F9807.TcDUT
{attribute 'GeneratedUsingTerminal: EM7004-0000-0016'}
{attribute addProperty BoxType "EM7004-0000-0016"}
{attribute addProperty Id "Latch_extern_validAT %I*BOOL1Set_counter_doneAT %I*BOOL1Status_of_input_AAT %I*BOOL1Status_of_input_BAT %I*BOOL1Status_of_input_gateAT %I*BOOL1Status_of_extern_latchAT %I*BOOL1TxPDO_ToggleAT %I*BOOL1Counter_valueAT %I*UINT2Latch_valueAT %I*UINT2"}
{attribute addProperty CRC "1802475527"}
{attribute addProperty Size "11"}
TYPE ENC_Inputs_Channel_6B6F9807 EXTENDS InputBase_8311D824 :
STRUCT
	{attribute addProperty Name "Latch_extern_valid"}
	Latch_extern_valid AT %I* : BOOL;
	{attribute addProperty Name "Set_counter_done"}
	Set_counter_done AT %I* : BOOL;
	{attribute addProperty Name "Status_of_input_A"}
	Status_of_input_A AT %I* : BOOL;
	{attribute addProperty Name "Status_of_input_B"}
	Status_of_input_B AT %I* : BOOL;
	{attribute addProperty Name "Status_of_input_gate"}
	Status_of_input_gate AT %I* : BOOL;
	{attribute addProperty Name "Status_of_extern_latch"}
	Status_of_extern_latch AT %I* : BOOL;
	{attribute addProperty Name "TxPDO_Toggle"}
	TxPDO_Toggle AT %I* : BOOL;
	{attribute addProperty Name "Counter_value"}
	Counter_value AT %I* : UINT;
	{attribute addProperty Name "Latch_value"}
	Latch_value AT %I* : UINT;
END_STRUCT
END_TYPE

// ---- DUTs/IO/PDOs/DI_Inputs_9882B618.TcDUT
{attribute 'GeneratedUsingTerminal: EM7004-0000-0017'}
{attribute addProperty BoxType "EM7004-0000-0017"}
{attribute addProperty Id "InputAT %I*Input_97D1F31316"}
{attribute addProperty CRC "2558703128"}
{attribute addProperty Size "16"}
TYPE DI_Inputs_9882B618 EXTENDS InputBase_8311D824 :
STRUCT
	{attribute addProperty Name "Input"}
	Input AT %I* : Input_97D1F313;
END_STRUCT
END_TYPE

// ---- DUTs/IO/PDOs/ENC_Inputs_Channel_E5B5E929.TcDUT
{attribute 'GeneratedUsingTerminal: EM7004-0000-0017'}
{attribute addProperty BoxType "EM7004-0000-0017"}
{attribute addProperty Id "StatusAT %I*Status_B4798D867Counter_valueAT %I*UINT2Latch_valueAT %I*UINT2"}
{attribute addProperty CRC "3853904169"}
{attribute addProperty Size "11"}
TYPE ENC_Inputs_Channel_E5B5E929 EXTENDS InputBase_8311D824 :
STRUCT
	{attribute addProperty Name "Status"}
	Status AT %I* : Status_B4798D86;
	{attribute addProperty Name "Counter_value"}
	Counter_value AT %I* : UINT;
	{attribute addProperty Name "Latch_value"}
	Latch_value AT %I* : UINT;
END_STRUCT
END_TYPE

// ---- DUTs/IO/PDOs/PLS_Inputs_65C9A3D6.TcDUT
{attribute 'GeneratedUsingTerminal: EM7004-0000-0017'}
{attribute addProperty BoxType "EM7004-0000-0017"}
{attribute addProperty Id "StatusAT %I*Status_882A150F2"}
{attribute addProperty CRC "1707713494"}
{attribute addProperty Size "2"}
TYPE PLS_Inputs_65C9A3D6 EXTENDS InputBase_8311D824 :
STRUCT
	{attribute addProperty Name "Status"}
	Status AT %I* : Status_882A150F;
END_STRUCT
END_TYPE

// ---- DUTs/IO/PDOs/DO_Outputs_47E26D6A.TcDUT
{attribute 'GeneratedUsingTerminal: EM7004-0000-0017'}
{attribute addProperty BoxType "EM7004-0000-0017"}
{attribute addProperty Id "OutputAT %Q*Output_FFFF807A16"}
{attribute addProperty CRC "1206021482"}
{attribute addProperty Size "16"}
TYPE DO_Outputs_47E26D6A EXTENDS OutputBase_10CEE7DE :
STRUCT
	{attribute addProperty Name "Output"}
	Output AT %Q* : Output_FFFF807A;
END_STRUCT
END_TYPE

// ---- DUTs/IO/PDOs/ENC_Outputs_Channel_2E82BC43.TcDUT
{attribute 'GeneratedUsingTerminal: EM7004-0000-0017'}
{attribute addProperty BoxType "EM7004-0000-0017"}
{attribute addProperty Id "ControlAT %Q*Control_F189B7373Set_counter_valueAT %Q*UINT2"}
{attribute addProperty CRC "780319811"}
{attribute addProperty Size "5"}
TYPE ENC_Outputs_Channel_2E82BC43 EXTENDS OutputBase_10CEE7DE :
STRUCT
	{attribute addProperty Name "Control"}
	Control AT %Q* : Control_F189B737;
	{attribute addProperty Name "Set_counter_value"}
	Set_counter_value AT %Q* : UINT;
END_STRUCT
END_TYPE

// ---- DUTs/IO/PDOs/PLS_Outputs_8EABC224.TcDUT
{attribute 'GeneratedUsingTerminal: EM7004-0000-0017'}
{attribute addProperty BoxType "EM7004-0000-0017"}
{attribute addProperty Id "ControlAT %Q*Control_17BA1FC21"}
{attribute addProperty CRC "2393621028"}
{attribute addProperty Size "1"}
TYPE PLS_Outputs_8EABC224 EXTENDS OutputBase_10CEE7DE :
STRUCT
	{attribute addProperty Name "Control"}
	Control AT %Q* : Control_17BA1FC2;
END_STRUCT
END_TYPE

// ---- DUTs/IO/PDOs/InfoData_E68C61CD.TcDUT
{attribute 'GeneratedUsingTerminal: IODEVICETYPE_ETHERCATPROT'}
{attribute addProperty BoxType "IODEVICETYPE_ETHERCATPROT"}
{attribute addProperty Id "ChangeCountAT %I*UINT2DevIdAT %I*UINT2AmsNetIdAT %I*AMSNETID6CfgSlaveCountAT %I*UINT2DcToTcTimeOffsetAT %I*LINT8DcToExtTimeOffsetAT %I*LINT8"}
{attribute addProperty CRC "3867959757"}
{attribute addProperty Size "28"}
TYPE InfoData_E68C61CD EXTENDS InputBase_8311D824 :
STRUCT
	{attribute addProperty Name "ChangeCount"}
	ChangeCount AT %I* : UINT;
	{attribute addProperty Name "DevId"}
	DevId AT %I* : UINT;
	{attribute addProperty Name "AmsNetId"}
	AmsNetId AT %I* : AMSNETID;
	{attribute addProperty Name "CfgSlaveCount"}
	CfgSlaveCount AT %I* : UINT;
	{attribute addProperty Name "DcToTcTimeOffset"}
	DcToTcTimeOffset AT %I* : LINT;
	{attribute addProperty Name "DcToExtTimeOffset"}
	DcToExtTimeOffset AT %I* : LINT;
END_STRUCT
END_TYPE

// ---- DUTs/IO/PDOs/InfoData_2A97D6CF.TcDUT
{attribute 'GeneratedUsingTerminal: IODEVICETYPE_ETHERCATPROT'}
{attribute addProperty BoxType "IODEVICETYPE_ETHERCATPROT"}
{attribute addProperty Id "ObjectIdAT %I*OTCID4StateAT %I*UINT2SlaveCountAT %I*UINT2"}
{attribute addProperty CRC "714593999"}
{attribute addProperty Size "8"}
TYPE InfoData_2A97D6CF EXTENDS InputBase_8311D824 :
STRUCT
	{attribute addProperty Name "ObjectId"}
	ObjectId AT %I* : OTCID;
	{attribute addProperty Name "State"}
	State AT %I* : UINT;
	{attribute addProperty Name "SlaveCount"}
	SlaveCount AT %I* : UINT;
END_STRUCT
END_TYPE

// ---- DUTs/IO/PDOs/Inputs_25A0042B.TcDUT
{attribute 'GeneratedUsingTerminal: IODEVICETYPE_ETHERCATPROT'}
{attribute addProperty BoxType "IODEVICETYPE_ETHERCATPROT"}
{attribute addProperty Id "SlaveCountAT %I*UINT2DevStateAT %I*UINT2Frm0StateAT %I*UINT2Frm0WcStateAT %I*UINT2Frm0InputToggleAT %I*UINT2Frm1StateAT %I*UINT2Frm1WcStateAT %I*UINT2Frm1InputToggleAT %I*UINT2Frm2StateAT %I*UINT2Frm2WcStateAT %I*UINT2Frm2InputToggleAT %I*UINT2Frm3StateAT %I*UINT2Frm3WcStateAT %I*UINT2Frm3InputToggleAT %I*UINT2Frm4StateAT %I*UINT2Frm4WcStateAT %I*UINT2Frm4InputToggleAT %I*UINT2Frm5StateAT %I*UINT2Frm5WcStateAT %I*UINT2Frm5InputToggleAT %I*UINT2Frm6StateAT %I*UINT2Frm6WcStateAT %I*UINT2Frm6InputToggleAT %I*UINT2Frm7StateAT %I*UINT2Frm7WcStateAT %I*UINT2Frm7InputToggleAT %I*UINT2Frm8StateAT %I*UINT2Frm8WcStateAT %I*UINT2Frm8InputToggleAT %I*UINT2Frm9StateAT %I*UINT2Frm9WcStateAT %I*UINT2Frm9InputToggleAT %I*UINT2Frm10StateAT %I*UINT2Frm10WcStateAT %I*UINT2Frm10InputToggleAT %I*UINT2Frm11StateAT %I*UINT2Frm11WcStateAT %I*UINT2Frm11InputToggleAT %I*UINT2Frm12StateAT %I*UINT2Frm12WcStateAT %I*UINT2Frm12InputToggleAT %I*UINT2Frm13StateAT %I*UINT2Frm13WcStateAT %I*UINT2Frm13InputToggleAT %I*UINT2Frm14StateAT %I*UINT2Frm14WcStateAT %I*UINT2Frm14InputToggleAT %I*UINT2Frm15StateAT %I*UINT2Frm15WcStateAT %I*UINT2Frm15InputToggleAT %I*UINT2Frm16StateAT %I*UINT2Frm16WcStateAT %I*UINT2Frm16InputToggleAT %I*UINT2Frm17StateAT %I*UINT2Frm17WcStateAT %I*UINT2Frm17InputToggleAT %I*UINT2Frm18StateAT %I*UINT2Frm18WcStateAT %I*UINT2Frm18InputToggleAT %I*UINT2Frm19StateAT %I*UINT2Frm19WcStateAT %I*UINT2Frm19InputToggleAT %I*UINT2Frm20StateAT %I*UINT2Frm20WcStateAT %I*UINT2Frm20InputToggleAT %I*UINT2Frm21StateAT %I*UINT2Frm21WcStateAT %I*UINT2Frm21InputToggleAT %I*UINT2Frm22StateAT %I*UINT2Frm22WcStateAT %I*UINT2Frm22InputToggleAT %I*UINT2Frm23StateAT %I*UINT2Frm23WcStateAT %I*UINT2Frm23InputToggleAT %I*UINT2Frm24StateAT %I*UINT2Frm24WcStateAT %I*UINT2Frm24InputToggleAT %I*UINT2Frm25StateAT %I*UINT2Frm25WcStateAT %I*UINT2Frm25InputToggleAT %I*UINT2"}
{attribute addProperty CRC "631243819"}
{attribute addProperty Size "160"}
TYPE Inputs_25A0042B EXTENDS InputBase_8311D824 :
STRUCT
	{attribute addProperty Name "SlaveCount"}
	SlaveCount AT %I* : UINT;
	{attribute addProperty Name "DevState"}
	DevState AT %I* : UINT;
	{attribute addProperty Name "Frm0State"}
	Frm0State AT %I* : UINT;
	{attribute addProperty Name "Frm0WcState"}
	Frm0WcState AT %I* : UINT;
	{attribute addProperty Name "Frm0InputToggle"}
	Frm0InputToggle AT %I* : UINT;
	{attribute addProperty Name "Frm1State"}
	Frm1State AT %I* : UINT;
	{attribute addProperty Name "Frm1WcState"}
	Frm1WcState AT %I* : UINT;
	{attribute addProperty Name "Frm1InputToggle"}
	Frm1InputToggle AT %I* : UINT;
	{attribute addProperty Name "Frm2State"}
	Frm2State AT %I* : UINT;
	{attribute addProperty Name "Frm2WcState"}
	Frm2WcState AT %I* : UINT;
	{attribute addProperty Name "Frm2InputToggle"}
	Frm2InputToggle AT %I* : UINT;
	{attribute addProperty Name "Frm3State"}
	Frm3State AT %I* : UINT;
	{attribute addProperty Name "Frm3WcState"}
	Frm3WcState AT %I* : UINT;
	{attribute addProperty Name "Frm3InputToggle"}
	Frm3InputToggle AT %I* : UINT;
	{attribute addProperty Name "Frm4State"}
	Frm4State AT %I* : UINT;
	{attribute addProperty Name "Frm4WcState"}
	Frm4WcState AT %I* : UINT;
	{attribute addProperty Name "Frm4InputToggle"}
	Frm4InputToggle AT %I* : UINT;
	{attribute addProperty Name "Frm5State"}
	Frm5State AT %I* : UINT;
	{attribute addProperty Name "Frm5WcState"}
	Frm5WcState AT %I* : UINT;
	{attribute addProperty Name "Frm5InputToggle"}
	Frm5InputToggle AT %I* : UINT;
	{attribute addProperty Name "Frm6State"}
	Frm6State AT %I* : UINT;
	{attribute addProperty Name "Frm6WcState"}
	Frm6WcState AT %I* : UINT;
	{attribute addProperty Name "Frm6InputToggle"}
	Frm6InputToggle AT %I* : UINT;
	{attribute addProperty Name "Frm7State"}
	Frm7State AT %I* : UINT;
	{attribute addProperty Name "Frm7WcState"}
	Frm7WcState AT %I* : UINT;
	{attribute addProperty Name "Frm7InputToggle"}
	Frm7InputToggle AT %I* : UINT;
	{attribute addProperty Name "Frm8State"}
	Frm8State AT %I* : UINT;
	{attribute addProperty Name "Frm8WcState"}
	Frm8WcState AT %I* : UINT;
	{attribute addProperty Name "Frm8InputToggle"}
	Frm8InputToggle AT %I* : UINT;
	{attribute addProperty Name "Frm9State"}
	Frm9State AT %I* : UINT;
	{attribute addProperty Name "Frm9WcState"}
	Frm9WcState AT %I* : UINT;
	{attribute addProperty Name "Frm9InputToggle"}
	Frm9InputToggle AT %I* : UINT;
	{attribute addProperty Name "Frm10State"}
	Frm10State AT %I* : UINT;
	{attribute addProperty Name "Frm10WcState"}
	Frm10WcState AT %I* : UINT;
	{attribute addProperty Name "Frm10InputToggle"}
	Frm10InputToggle AT %I* : UINT;
	{attribute addProperty Name "Frm11State"}
	Frm11State AT %I* : UINT;
	{attribute addProperty Name "Frm11WcState"}
	Frm11WcState AT %I* : UINT;
	{attribute addProperty Name "Frm11InputToggle"}
	Frm11InputToggle AT %I* : UINT;
	{attribute addProperty Name "Frm12State"}
	Frm12State AT %I* : UINT;
	{attribute addProperty Name "Frm12WcState"}
	Frm12WcState AT %I* : UINT;
	{attribute addProperty Name "Frm12InputToggle"}
	Frm12InputToggle AT %I* : UINT;
	{attribute addProperty Name "Frm13State"}
	Frm13State AT %I* : UINT;
	{attribute addProperty Name "Frm13WcState"}
	Frm13WcState AT %I* : UINT;
	{attribute addProperty Name "Frm13InputToggle"}
	Frm13InputToggle AT %I* : UINT;
	{attribute addProperty Name "Frm14State"}
	Frm14State AT %I* : UINT;
	{attribute addProperty Name "Frm14WcState"}
	Frm14WcState AT %I* : UINT;
	{attribute addProperty Name "Frm14InputToggle"}
	Frm14InputToggle AT %I* : UINT;
	{attribute addProperty Name "Frm15State"}
	Frm15State AT %I* : UINT;
	{attribute addProperty Name "Frm15WcState"}
	Frm15WcState AT %I* : UINT;
	{attribute addProperty Name "Frm15InputToggle"}
	Frm15InputToggle AT %I* : UINT;
	{attribute addProperty Name "Frm16State"}
	Frm16State AT %I* : UINT;
	{attribute addProperty Name "Frm16WcState"}
	Frm16WcState AT %I* : UINT;
	{attribute addProperty Name "Frm16InputToggle"}
	Frm16InputToggle AT %I* : UINT;
	{attribute addProperty Name "Frm17State"}
	Frm17State AT %I* : UINT;
	{attribute addProperty Name "Frm17WcState"}
	Frm17WcState AT %I* : UINT;
	{attribute addProperty Name "Frm17InputToggle"}
	Frm17InputToggle AT %I* : UINT;
	{attribute addProperty Name "Frm18State"}
	Frm18State AT %I* : UINT;
	{attribute addProperty Name "Frm18WcState"}
	Frm18WcState AT %I* : UINT;
	{attribute addProperty Name "Frm18InputToggle"}
	Frm18InputToggle AT %I* : UINT;
	{attribute addProperty Name "Frm19State"}
	Frm19State AT %I* : UINT;
	{attribute addProperty Name "Frm19WcState"}
	Frm19WcState AT %I* : UINT;
	{attribute addProperty Name "Frm19InputToggle"}
	Frm19InputToggle AT %I* : UINT;
	{attribute addProperty Name "Frm20State"}
	Frm20State AT %I* : UINT;
	{attribute addProperty Name "Frm20WcState"}
	Frm20WcState AT %I* : UINT;
	{attribute addProperty Name "Frm20InputToggle"}
	Frm20InputToggle AT %I* : UINT;
	{attribute addProperty Name "Frm21State"}
	Frm21State AT %I* : UINT;
	{attribute addProperty Name "Frm21WcState"}
	Frm21WcState AT %I* : UINT;
	{attribute addProperty Name "Frm21InputToggle"}
	Frm21InputToggle AT %I* : UINT;
	{attribute addProperty Name "Frm22State"}
	Frm22State AT %I* : UINT;
	{attribute addProperty Name "Frm22WcState"}
	Frm22WcState AT %I* : UINT;
	{attribute addProperty Name "Frm22InputToggle"}
	Frm22InputToggle AT %I* : UINT;
	{attribute addProperty Name "Frm23State"}
	Frm23State AT %I* : UINT;
	{attribute addProperty Name "Frm23WcState"}
	Frm23WcState AT %I* : UINT;
	{attribute addProperty Name "Frm23InputToggle"}
	Frm23InputToggle AT %I* : UINT;
	{attribute addProperty Name "Frm24State"}
	Frm24State AT %I* : UINT;
	{attribute addProperty Name "Frm24WcState"}
	Frm24WcState AT %I* : UINT;
	{attribute addProperty Name "Frm24InputToggle"}
	Frm24InputToggle AT %I* : UINT;
	{attribute addProperty Name "Frm25State"}
	Frm25State AT %I* : UINT;
	{attribute addProperty Name "Frm25WcState"}
	Frm25WcState AT %I* : UINT;
	{attribute addProperty Name "Frm25InputToggle"}
	Frm25InputToggle AT %I* : UINT;
END_STRUCT
END_TYPE

// ---- DUTs/IO/PDOs/Outputs_2397A10E.TcDUT
{attribute 'GeneratedUsingTerminal: IODEVICETYPE_ETHERCATPROT'}
{attribute addProperty BoxType "IODEVICETYPE_ETHERCATPROT"}
{attribute addProperty Id "DevCtrlAT %Q*UINT2Frm0CtrlAT %Q*UINT2Frm0WcCtrlAT %Q*UINT2Frm1CtrlAT %Q*UINT2Frm1WcCtrlAT %Q*UINT2Frm2CtrlAT %Q*UINT2Frm2WcCtrlAT %Q*UINT2Frm3CtrlAT %Q*UINT2Frm3WcCtrlAT %Q*UINT2Frm4CtrlAT %Q*UINT2Frm4WcCtrlAT %Q*UINT2Frm5CtrlAT %Q*UINT2Frm5WcCtrlAT %Q*UINT2Frm6CtrlAT %Q*UINT2Frm6WcCtrlAT %Q*UINT2Frm7CtrlAT %Q*UINT2Frm7WcCtrlAT %Q*UINT2Frm8CtrlAT %Q*UINT2Frm8WcCtrlAT %Q*UINT2Frm9CtrlAT %Q*UINT2Frm9WcCtrlAT %Q*UINT2Frm10CtrlAT %Q*UINT2Frm10WcCtrlAT %Q*UINT2Frm11CtrlAT %Q*UINT2Frm11WcCtrlAT %Q*UINT2Frm12CtrlAT %Q*UINT2Frm12WcCtrlAT %Q*UINT2Frm13CtrlAT %Q*UINT2Frm13WcCtrlAT %Q*UINT2Frm14CtrlAT %Q*UINT2Frm14WcCtrlAT %Q*UINT2Frm15CtrlAT %Q*UINT2Frm15WcCtrlAT %Q*UINT2Frm16CtrlAT %Q*UINT2Frm16WcCtrlAT %Q*UINT2Frm17CtrlAT %Q*UINT2Frm17WcCtrlAT %Q*UINT2Frm18CtrlAT %Q*UINT2Frm18WcCtrlAT %Q*UINT2Frm19CtrlAT %Q*UINT2Frm19WcCtrlAT %Q*UINT2Frm20CtrlAT %Q*UINT2Frm20WcCtrlAT %Q*UINT2Frm21CtrlAT %Q*UINT2Frm21WcCtrlAT %Q*UINT2Frm22CtrlAT %Q*UINT2Frm22WcCtrlAT %Q*UINT2Frm23CtrlAT %Q*UINT2Frm23WcCtrlAT %Q*UINT2Frm24CtrlAT %Q*UINT2Frm24WcCtrlAT %Q*UINT2Frm25CtrlAT %Q*UINT2Frm25WcCtrlAT %Q*UINT2"}
{attribute addProperty CRC "597139726"}
{attribute addProperty Size "106"}
TYPE Outputs_2397A10E EXTENDS OutputBase_10CEE7DE :
STRUCT
	{attribute addProperty Name "DevCtrl"}
	DevCtrl AT %Q* : UINT;
	{attribute addProperty Name "Frm0Ctrl"}
	Frm0Ctrl AT %Q* : UINT;
	{attribute addProperty Name "Frm0WcCtrl"}
	Frm0WcCtrl AT %Q* : UINT;
	{attribute addProperty Name "Frm1Ctrl"}
	Frm1Ctrl AT %Q* : UINT;
	{attribute addProperty Name "Frm1WcCtrl"}
	Frm1WcCtrl AT %Q* : UINT;
	{attribute addProperty Name "Frm2Ctrl"}
	Frm2Ctrl AT %Q* : UINT;
	{attribute addProperty Name "Frm2WcCtrl"}
	Frm2WcCtrl AT %Q* : UINT;
	{attribute addProperty Name "Frm3Ctrl"}
	Frm3Ctrl AT %Q* : UINT;
	{attribute addProperty Name "Frm3WcCtrl"}
	Frm3WcCtrl AT %Q* : UINT;
	{attribute addProperty Name "Frm4Ctrl"}
	Frm4Ctrl AT %Q* : UINT;
	{attribute addProperty Name "Frm4WcCtrl"}
	Frm4WcCtrl AT %Q* : UINT;
	{attribute addProperty Name "Frm5Ctrl"}
	Frm5Ctrl AT %Q* : UINT;
	{attribute addProperty Name "Frm5WcCtrl"}
	Frm5WcCtrl AT %Q* : UINT;
	{attribute addProperty Name "Frm6Ctrl"}
	Frm6Ctrl AT %Q* : UINT;
	{attribute addProperty Name "Frm6WcCtrl"}
	Frm6WcCtrl AT %Q* : UINT;
	{attribute addProperty Name "Frm7Ctrl"}
	Frm7Ctrl AT %Q* : UINT;
	{attribute addProperty Name "Frm7WcCtrl"}
	Frm7WcCtrl AT %Q* : UINT;
	{attribute addProperty Name "Frm8Ctrl"}
	Frm8Ctrl AT %Q* : UINT;
	{attribute addProperty Name "Frm8WcCtrl"}
	Frm8WcCtrl AT %Q* : UINT;
	{attribute addProperty Name "Frm9Ctrl"}
	Frm9Ctrl AT %Q* : UINT;
	{attribute addProperty Name "Frm9WcCtrl"}
	Frm9WcCtrl AT %Q* : UINT;
	{attribute addProperty Name "Frm10Ctrl"}
	Frm10Ctrl AT %Q* : UINT;
	{attribute addProperty Name "Frm10WcCtrl"}
	Frm10WcCtrl AT %Q* : UINT;
	{attribute addProperty Name "Frm11Ctrl"}
	Frm11Ctrl AT %Q* : UINT;
	{attribute addProperty Name "Frm11WcCtrl"}
	Frm11WcCtrl AT %Q* : UINT;
	{attribute addProperty Name "Frm12Ctrl"}
	Frm12Ctrl AT %Q* : UINT;
	{attribute addProperty Name "Frm12WcCtrl"}
	Frm12WcCtrl AT %Q* : UINT;
	{attribute addProperty Name "Frm13Ctrl"}
	Frm13Ctrl AT %Q* : UINT;
	{attribute addProperty Name "Frm13WcCtrl"}
	Frm13WcCtrl AT %Q* : UINT;
	{attribute addProperty Name "Frm14Ctrl"}
	Frm14Ctrl AT %Q* : UINT;
	{attribute addProperty Name "Frm14WcCtrl"}
	Frm14WcCtrl AT %Q* : UINT;
	{attribute addProperty Name "Frm15Ctrl"}
	Frm15Ctrl AT %Q* : UINT;
	{attribute addProperty Name "Frm15WcCtrl"}
	Frm15WcCtrl AT %Q* : UINT;
	{attribute addProperty Name "Frm16Ctrl"}
	Frm16Ctrl AT %Q* : UINT;
	{attribute addProperty Name "Frm16WcCtrl"}
	Frm16WcCtrl AT %Q* : UINT;
	{attribute addProperty Name "Frm17Ctrl"}
	Frm17Ctrl AT %Q* : UINT;
	{attribute addProperty Name "Frm17WcCtrl"}
	Frm17WcCtrl AT %Q* : UINT;
	{attribute addProperty Name "Frm18Ctrl"}
	Frm18Ctrl AT %Q* : UINT;
	{attribute addProperty Name "Frm18WcCtrl"}
	Frm18WcCtrl AT %Q* : UINT;
	{attribute addProperty Name "Frm19Ctrl"}
	Frm19Ctrl AT %Q* : UINT;
	{attribute addProperty Name "Frm19WcCtrl"}
	Frm19WcCtrl AT %Q* : UINT;
	{attribute addProperty Name "Frm20Ctrl"}
	Frm20Ctrl AT %Q* : UINT;
	{attribute addProperty Name "Frm20WcCtrl"}
	Frm20WcCtrl AT %Q* : UINT;
	{attribute addProperty Name "Frm21Ctrl"}
	Frm21Ctrl AT %Q* : UINT;
	{attribute addProperty Name "Frm21WcCtrl"}
	Frm21WcCtrl AT %Q* : UINT;
	{attribute addProperty Name "Frm22Ctrl"}
	Frm22Ctrl AT %Q* : UINT;
	{attribute addProperty Name "Frm22WcCtrl"}
	Frm22WcCtrl AT %Q* : UINT;
	{attribute addProperty Name "Frm23Ctrl"}
	Frm23Ctrl AT %Q* : UINT;
	{attribute addProperty Name "Frm23WcCtrl"}
	Frm23WcCtrl AT %Q* : UINT;
	{attribute addProperty Name "Frm24Ctrl"}
	Frm24Ctrl AT %Q* : UINT;
	{attribute addProperty Name "Frm24WcCtrl"}
	Frm24WcCtrl AT %Q* : UINT;
	{attribute addProperty Name "Frm25Ctrl"}
	Frm25Ctrl AT %Q* : UINT;
	{attribute addProperty Name "Frm25WcCtrl"}
	Frm25WcCtrl AT %Q* : UINT;
END_STRUCT
END_TYPE

// ---- DUTs/IO/Boxes/EK1100_1FC0878B.TcDUT
{attribute 'GeneratedUsingTerminal: EK1100-0000-0018'}
{attribute addProperty BoxType "EK1100-0000-0018"}
{attribute addProperty Description "EK1100 EtherCAT Coupler (2A E-Bus)"}
{attribute addProperty Physics "YKY"}
{attribute addProperty Id "InfoDataAT %I*InfoData_6F19DB2B2"}
{attribute addProperty CRC "532711307"}
{attribute addProperty Size "2"}
TYPE EK1100_1FC0878B EXTENDS EtcSlaveBoxBase_77A0E4A7 :
STRUCT
	{attribute addProperty Name "InfoData"}
	InfoData : InfoData_6F19DB2B;
END_STRUCT
END_TYPE

// ---- DUTs/IO/Boxes/EK1122_1FC0878B.TcDUT
{attribute 'GeneratedUsingTerminal: EK1122-0000-0018'}
{attribute addProperty BoxType "EK1122-0000-0018"}
{attribute addProperty Description "EK1122 2 port EtherCAT junction"}
{attribute addProperty Physics "KYKY"}
{attribute addProperty Id "InfoDataAT %I*InfoData_6F19DB2B2"}
{attribute addProperty CRC "532711307"}
{attribute addProperty Size "2"}
TYPE EK1122_1FC0878B EXTENDS EtcSlaveTerminalBase_947E5A46 :
STRUCT
	{attribute addProperty Name "InfoData"}
	InfoData : InfoData_6F19DB2B;
END_STRUCT
END_TYPE

// ---- DUTs/IO/Boxes/EM2042_2B6483BD.TcDUT
{attribute 'GeneratedUsingTerminal: EM2042-0000-0016'}
{attribute addProperty BoxType "EM2042-0000-0016"}
{attribute addProperty Description "EM2042 16Ch. Dig. Output 24V, 0.5A, D-Sub connection"}
{attribute addProperty Physics "KK"}
{attribute addProperty Id "Channel_1AT %Q*Channel_42CA91F71Channel_2AT %Q*Channel_42CA91F71Channel_3AT %Q*Channel_42CA91F71Channel_4AT %Q*Channel_42CA91F71Channel_5AT %Q*Channel_42CA91F71Channel_6AT %Q*Channel_42CA91F71Channel_7AT %Q*Channel_42CA91F71Channel_8AT %Q*Channel_42CA91F71Channel_9AT %Q*Channel_42CA91F71Channel_10AT %Q*Channel_42CA91F71Channel_11AT %Q*Channel_42CA91F71Channel_12AT %Q*Channel_42CA91F71Channel_13AT %Q*Channel_42CA91F71Channel_14AT %Q*Channel_42CA91F71Channel_15AT %Q*Channel_42CA91F71Channel_16AT %Q*Channel_42CA91F71WcStateAT %I*WcState_0B2B16F91InfoDataAT %I*InfoData_6F19DB2B2"}
{attribute addProperty CRC "728007613"}
{attribute addProperty Size "19"}
TYPE EM2042_2B6483BD EXTENDS EtcSlaveTerminalBase_947E5A46 :
STRUCT
	{attribute addProperty Name "Channel_1"}
	Channel_1 : Channel_42CA91F7;
	{attribute addProperty Name "Channel_2"}
	Channel_2 : Channel_42CA91F7;
	{attribute addProperty Name "Channel_3"}
	Channel_3 : Channel_42CA91F7;
	{attribute addProperty Name "Channel_4"}
	Channel_4 : Channel_42CA91F7;
	{attribute addProperty Name "Channel_5"}
	Channel_5 : Channel_42CA91F7;
	{attribute addProperty Name "Channel_6"}
	Channel_6 : Channel_42CA91F7;
	{attribute addProperty Name "Channel_7"}
	Channel_7 : Channel_42CA91F7;
	{attribute addProperty Name "Channel_8"}
	Channel_8 : Channel_42CA91F7;
	{attribute addProperty Name "Channel_9"}
	Channel_9 : Channel_42CA91F7;
	{attribute addProperty Name "Channel_10"}
	Channel_10 : Channel_42CA91F7;
	{attribute addProperty Name "Channel_11"}
	Channel_11 : Channel_42CA91F7;
	{attribute addProperty Name "Channel_12"}
	Channel_12 : Channel_42CA91F7;
	{attribute addProperty Name "Channel_13"}
	Channel_13 : Channel_42CA91F7;
	{attribute addProperty Name "Channel_14"}
	Channel_14 : Channel_42CA91F7;
	{attribute addProperty Name "Channel_15"}
	Channel_15 : Channel_42CA91F7;
	{attribute addProperty Name "Channel_16"}
	Channel_16 : Channel_42CA91F7;
	{attribute addProperty Name "WcState"}
	WcState : WcState_0B2B16F9;
	{attribute addProperty Name "InfoData"}
	InfoData : InfoData_6F19DB2B;
END_STRUCT
END_TYPE

// ---- DUTs/IO/Boxes/EM3701_AB0D469D.TcDUT
{attribute 'GeneratedUsingTerminal: EM3701-0000-0016'}
{attribute addProperty BoxType "EM3701-0000-0016"}
{attribute addProperty Description "EM3701, 1Ch. differential pressure measuring terminal 100hPa (100mbar)"}
{attribute addProperty Physics "KK"}
{attribute addProperty Id "AI_InputsAT %I*AI_Inputs_5AF6604E8WcStateAT %I*WcState_9091E0EB2InfoDataAT %I*InfoData_32EB74EA10"}
{attribute addProperty CRC "2869773981"}
{attribute addProperty Size "20"}
TYPE EM3701_AB0D469D EXTENDS EtcSlaveTerminalBase_947E5A46 :
STRUCT
	{attribute addProperty Name "AI_Inputs"}
	AI_Inputs : AI_Inputs_5AF6604E;
	{attribute addProperty Name "WcState"}
	WcState : WcState_9091E0EB;
	{attribute addProperty Name "InfoData"}
	InfoData : InfoData_32EB74EA;
END_STRUCT
END_TYPE

// ---- DUTs/IO/Boxes/EM3702_FDD84FD8.TcDUT
{attribute 'GeneratedUsingTerminal: EM3702-0000-0016'}
{attribute addProperty BoxType "EM3702-0000-0016"}
{attribute addProperty Description "EM3702  2Ch. relative pressure measuring terminal 7,500 hPa (7.5 bar)"}
{attribute addProperty Physics "KK"}
{attribute addProperty Id "AI_Input_Channel_1AT %I*AI_Input_Channel_5AF6604E8AI_Input_Channel_2AT %I*AI_Input_Channel_5AF6604E8WcStateAT %I*WcState_9091E0EB2InfoDataAT %I*InfoData_32EB74EA10"}
{attribute addProperty CRC "4258811864"}
{attribute addProperty Size "28"}
TYPE EM3702_FDD84FD8 EXTENDS EtcSlaveTerminalBase_947E5A46 :
STRUCT
	{attribute addProperty Name "AI_Input_Channel_1"}
	AI_Input_Channel_1 : AI_Input_Channel_5AF6604E;
	{attribute addProperty Name "AI_Input_Channel_2"}
	AI_Input_Channel_2 : AI_Input_Channel_5AF6604E;
	{attribute addProperty Name "WcState"}
	WcState : WcState_9091E0EB;
	{attribute addProperty Name "InfoData"}
	InfoData : InfoData_32EB74EA;
END_STRUCT
END_TYPE

// ---- DUTs/IO/Boxes/EM3712_FDD84FD8.TcDUT
{attribute 'GeneratedUsingTerminal: EM3712-0000-0016'}
{attribute addProperty BoxType "EM3712-0000-0016"}
{attribute addProperty Description "EM3712  2Ch relative pressure measuring terminal -1,000...+1,000 hPa (-1...+1 bar)"}
{attribute addProperty Physics "KK"}
{attribute addProperty Id "AI_Input_Channel_1AT %I*AI_Input_Channel_5AF6604E8AI_Input_Channel_2AT %I*AI_Input_Channel_5AF6604E8WcStateAT %I*WcState_9091E0EB2InfoDataAT %I*InfoData_32EB74EA10"}
{attribute addProperty CRC "4258811864"}
{attribute addProperty Size "28"}
TYPE EM3712_FDD84FD8 EXTENDS EtcSlaveTerminalBase_947E5A46 :
STRUCT
	{attribute addProperty Name "AI_Input_Channel_1"}
	AI_Input_Channel_1 : AI_Input_Channel_5AF6604E;
	{attribute addProperty Name "AI_Input_Channel_2"}
	AI_Input_Channel_2 : AI_Input_Channel_5AF6604E;
	{attribute addProperty Name "WcState"}
	WcState : WcState_9091E0EB;
	{attribute addProperty Name "InfoData"}
	InfoData : InfoData_32EB74EA;
END_STRUCT
END_TYPE

// ---- DUTs/IO/Boxes/EM7004_866015E1.TcDUT
{attribute 'GeneratedUsingTerminal: EM7004-0000-9995'}
{attribute addProperty BoxType "EM7004-0000-9995"}
{attribute addProperty Description "EM7004 4-Axis Interface Unit"}
{attribute addProperty Physics "KK"}
{attribute addProperty Id "DigitalAT %I*Digital_BD004D6F16Encoder_Channel_1AT %I*Encoder_Channel_2E4EA2136Encoder_Channel_2AT %I*Encoder_Channel_2E4EA2136Encoder_Channel_3AT %I*Encoder_Channel_2E4EA2136Encoder_Channel_4AT %I*Encoder_Channel_2E4EA2136Digital_1AT %Q*Digital_A7E1DFAB16Analog_Channel_1AT %Q*Analog_Channel_5F9B7EA62Analog_Channel_2AT %Q*Analog_Channel_5F9B7EA62Analog_Channel_3AT %Q*Analog_Channel_5F9B7EA62Analog_Channel_4AT %Q*Analog_Channel_5F9B7EA62Encoder_Channel_1_1AT %Q*Encoder_Channel_B7999E144Encoder_Channel_2_1AT %Q*Encoder_Channel_B7999E144Encoder_Channel_3_1AT %Q*Encoder_Channel_B7999E144Encoder_Channel_4_1AT %Q*Encoder_Channel_B7999E144WcStateAT %I*WcState_9091E0EB2InfoDataAT %I*InfoData_32EB74EA10"}
{attribute addProperty CRC "2254444001"}
{attribute addProperty Size "92"}
TYPE EM7004_866015E1 EXTENDS EtcSlaveTerminalBase_947E5A46 :
STRUCT
	{attribute addProperty Name "Digital"}
	Digital : Digital_BD004D6F;
	{attribute addProperty Name "Encoder_Channel_1"}
	Encoder_Channel_1 : Encoder_Channel_2E4EA213;
	{attribute addProperty Name "Encoder_Channel_2"}
	Encoder_Channel_2 : Encoder_Channel_2E4EA213;
	{attribute addProperty Name "Encoder_Channel_3"}
	Encoder_Channel_3 : Encoder_Channel_2E4EA213;
	{attribute addProperty Name "Encoder_Channel_4"}
	Encoder_Channel_4 : Encoder_Channel_2E4EA213;
	{attribute addProperty Name "Digital_1"}
	Digital_1 : Digital_A7E1DFAB;
	{attribute addProperty Name "Analog_Channel_1"}
	Analog_Channel_1 : Analog_Channel_5F9B7EA6;
	{attribute addProperty Name "Analog_Channel_2"}
	Analog_Channel_2 : Analog_Channel_5F9B7EA6;
	{attribute addProperty Name "Analog_Channel_3"}
	Analog_Channel_3 : Analog_Channel_5F9B7EA6;
	{attribute addProperty Name "Analog_Channel_4"}
	Analog_Channel_4 : Analog_Channel_5F9B7EA6;
	{attribute addProperty Name "Encoder_Channel_1_1"}
	Encoder_Channel_1_1 : Encoder_Channel_B7999E14;
	{attribute addProperty Name "Encoder_Channel_2_1"}
	Encoder_Channel_2_1 : Encoder_Channel_B7999E14;
	{attribute addProperty Name "Encoder_Channel_3_1"}
	Encoder_Channel_3_1 : Encoder_Channel_B7999E14;
	{attribute addProperty Name "Encoder_Channel_4_1"}
	Encoder_Channel_4_1 : Encoder_Channel_B7999E14;
	{attribute addProperty Name "WcState"}
	WcState : WcState_9091E0EB;
	{attribute addProperty Name "InfoData"}
	InfoData : InfoData_32EB74EA;
END_STRUCT
END_TYPE

// ---- DUTs/IO/Boxes/EM7004_7586CC95.TcDUT
{attribute 'GeneratedUsingTerminal: EM7004-0000-9996'}
{attribute addProperty BoxType "EM7004-0000-9996"}
{attribute addProperty Description "EM7004 4-Axis Interface Unit"}
{attribute addProperty Physics "KK"}
{attribute addProperty Id "DI_InputsAT %I*DI_Inputs_BD004D6F16ENC_Inputs_Channel_1AT %I*ENC_Inputs_Channel_69C51E8E10ENC_Inputs_Channel_2AT %I*ENC_Inputs_Channel_69C51E8E10ENC_Inputs_Channel_3AT %I*ENC_Inputs_Channel_69C51E8E10ENC_Inputs_Channel_4AT %I*ENC_Inputs_Channel_69C51E8E10PLS_InputsAT %I*PLS_Inputs_5A35B63D2DO_OutputsAT %Q*DO_Outputs_A7E1DFAB16AO_Outputs_Channel_1AT %Q*AO_Output_Channel_BA7EBB7C2AO_Outputs_Channel_2AT %Q*AO_Output_Channel_BA7EBB7C2AO_Outputs_Channel_3AT %Q*AO_Output_Channel_BA7EBB7C2AO_Outputs_Channel_4AT %Q*AO_Output_Channel_BA7EBB7C2ENC_Outputs_Channel_1AT %Q*ENC_Outputs_Channel_DC4E290B5ENC_Outputs_Channel_2AT %Q*ENC_Outputs_Channel_DC4E290B5ENC_Outputs_Channel_3AT %Q*ENC_Outputs_Channel_DC4E290B5ENC_Outputs_Channel_4AT %Q*ENC_Outputs_Channel_DC4E290B5PLS_OutputsAT %Q*PLS_Outputs_AFB7DAF51WcStateAT %I*WcState_9091E0EB2InfoDataAT %I*InfoData_32EB74EA10"}
{attribute addProperty CRC "1971768469"}
{attribute addProperty Size "115"}
TYPE EM7004_7586CC95 EXTENDS EtcSlaveTerminalBase_947E5A46 :
STRUCT
	{attribute addProperty Name "DI_Inputs"}
	DI_Inputs : DI_Inputs_BD004D6F;
	{attribute addProperty Name "ENC_Inputs_Channel_1"}
	ENC_Inputs_Channel_1 : ENC_Inputs_Channel_69C51E8E;
	{attribute addProperty Name "ENC_Inputs_Channel_2"}
	ENC_Inputs_Channel_2 : ENC_Inputs_Channel_69C51E8E;
	{attribute addProperty Name "ENC_Inputs_Channel_3"}
	ENC_Inputs_Channel_3 : ENC_Inputs_Channel_69C51E8E;
	{attribute addProperty Name "ENC_Inputs_Channel_4"}
	ENC_Inputs_Channel_4 : ENC_Inputs_Channel_69C51E8E;
	{attribute addProperty Name "PLS_Inputs"}
	PLS_Inputs : PLS_Inputs_5A35B63D;
	{attribute addProperty Name "DO_Outputs"}
	DO_Outputs : DO_Outputs_A7E1DFAB;
	{attribute addProperty Name "AO_Outputs_Channel_1"}
	AO_Outputs_Channel_1 : AO_Output_Channel_BA7EBB7C;
	{attribute addProperty Name "AO_Outputs_Channel_2"}
	AO_Outputs_Channel_2 : AO_Output_Channel_BA7EBB7C;
	{attribute addProperty Name "AO_Outputs_Channel_3"}
	AO_Outputs_Channel_3 : AO_Output_Channel_BA7EBB7C;
	{attribute addProperty Name "AO_Outputs_Channel_4"}
	AO_Outputs_Channel_4 : AO_Output_Channel_BA7EBB7C;
	{attribute addProperty Name "ENC_Outputs_Channel_1"}
	ENC_Outputs_Channel_1 : ENC_Outputs_Channel_DC4E290B;
	{attribute addProperty Name "ENC_Outputs_Channel_2"}
	ENC_Outputs_Channel_2 : ENC_Outputs_Channel_DC4E290B;
	{attribute addProperty Name "ENC_Outputs_Channel_3"}
	ENC_Outputs_Channel_3 : ENC_Outputs_Channel_DC4E290B;
	{attribute addProperty Name "ENC_Outputs_Channel_4"}
	ENC_Outputs_Channel_4 : ENC_Outputs_Channel_DC4E290B;
	{attribute addProperty Name "PLS_Outputs"}
	PLS_Outputs : PLS_Outputs_AFB7DAF5;
	{attribute addProperty Name "WcState"}
	WcState : WcState_9091E0EB;
	{attribute addProperty Name "InfoData"}
	InfoData : InfoData_32EB74EA;
END_STRUCT
END_TYPE

// ---- DUTs/IO/Boxes/EM7004_5FA1DD22.TcDUT
{attribute 'GeneratedUsingTerminal: EM7004-0000-0016'}
{attribute addProperty BoxType "EM7004-0000-0016"}
{attribute addProperty Description "EM7004 4-Axis Interface Unit"}
{attribute addProperty Physics "KK"}
{attribute addProperty Id "DI_InputsAT %I*DI_Inputs_BD004D6F16ENC_Inputs_Channel_1AT %I*ENC_Inputs_Channel_6B6F980711ENC_Inputs_Channel_2AT %I*ENC_Inputs_Channel_6B6F980711ENC_Inputs_Channel_3AT %I*ENC_Inputs_Channel_6B6F980711ENC_Inputs_Channel_4AT %I*ENC_Inputs_Channel_6B6F980711PLS_InputsAT %I*PLS_Inputs_5A35B63D2DO_OutputsAT %Q*DO_Outputs_A7E1DFAB16AO_Outputs_Channel_1AT %Q*AO_Output_Channel_BA7EBB7C2AO_Outputs_Channel_2AT %Q*AO_Output_Channel_BA7EBB7C2AO_Outputs_Channel_3AT %Q*AO_Output_Channel_BA7EBB7C2AO_Outputs_Channel_4AT %Q*AO_Output_Channel_BA7EBB7C2ENC_Outputs_Channel_1AT %Q*ENC_Outputs_Channel_DC4E290B5ENC_Outputs_Channel_2AT %Q*ENC_Outputs_Channel_DC4E290B5ENC_Outputs_Channel_3AT %Q*ENC_Outputs_Channel_DC4E290B5ENC_Outputs_Channel_4AT %Q*ENC_Outputs_Channel_DC4E290B5PLS_OutputsAT %Q*PLS_Outputs_AFB7DAF51WcStateAT %I*WcState_9091E0EB2InfoDataAT %I*InfoData_32EB74EA10"}
{attribute addProperty CRC "1604443426"}
{attribute addProperty Size "119"}
TYPE EM7004_5FA1DD22 EXTENDS EtcSlaveTerminalBase_947E5A46 :
STRUCT
	{attribute addProperty Name "DI_Inputs"}
	DI_Inputs : DI_Inputs_BD004D6F;
	{attribute addProperty Name "ENC_Inputs_Channel_1"}
	ENC_Inputs_Channel_1 : ENC_Inputs_Channel_6B6F9807;
	{attribute addProperty Name "ENC_Inputs_Channel_2"}
	ENC_Inputs_Channel_2 : ENC_Inputs_Channel_6B6F9807;
	{attribute addProperty Name "ENC_Inputs_Channel_3"}
	ENC_Inputs_Channel_3 : ENC_Inputs_Channel_6B6F9807;
	{attribute addProperty Name "ENC_Inputs_Channel_4"}
	ENC_Inputs_Channel_4 : ENC_Inputs_Channel_6B6F9807;
	{attribute addProperty Name "PLS_Inputs"}
	PLS_Inputs : PLS_Inputs_5A35B63D;
	{attribute addProperty Name "DO_Outputs"}
	DO_Outputs : DO_Outputs_A7E1DFAB;
	{attribute addProperty Name "AO_Outputs_Channel_1"}
	AO_Outputs_Channel_1 : AO_Output_Channel_BA7EBB7C;
	{attribute addProperty Name "AO_Outputs_Channel_2"}
	AO_Outputs_Channel_2 : AO_Output_Channel_BA7EBB7C;
	{attribute addProperty Name "AO_Outputs_Channel_3"}
	AO_Outputs_Channel_3 : AO_Output_Channel_BA7EBB7C;
	{attribute addProperty Name "AO_Outputs_Channel_4"}
	AO_Outputs_Channel_4 : AO_Output_Channel_BA7EBB7C;
	{attribute addProperty Name "ENC_Outputs_Channel_1"}
	ENC_Outputs_Channel_1 : ENC_Outputs_Channel_DC4E290B;
	{attribute addProperty Name "ENC_Outputs_Channel_2"}
	ENC_Outputs_Channel_2 : ENC_Outputs_Channel_DC4E290B;
	{attribute addProperty Name "ENC_Outputs_Channel_3"}
	ENC_Outputs_Channel_3 : ENC_Outputs_Channel_DC4E290B;
	{attribute addProperty Name "ENC_Outputs_Channel_4"}
	ENC_Outputs_Channel_4 : ENC_Outputs_Channel_DC4E290B;
	{attribute addProperty Name "PLS_Outputs"}
	PLS_Outputs : PLS_Outputs_AFB7DAF5;
	{attribute addProperty Name "WcState"}
	WcState : WcState_9091E0EB;
	{attribute addProperty Name "InfoData"}
	InfoData : InfoData_32EB74EA;
END_STRUCT
END_TYPE

// ---- DUTs/IO/Boxes/EM7004_0F97553F.TcDUT
{attribute 'GeneratedUsingTerminal: EM7004-0000-0017'}
{attribute addProperty BoxType "EM7004-0000-0017"}
{attribute addProperty Description "EM7004 4-Axis Interface Unit"}
{attribute addProperty Physics "KK"}
{attribute addProperty Id "DI_InputsAT %I*DI_Inputs_9882B61816ENC_Inputs_Channel_1AT %I*ENC_Inputs_Channel_E5B5E92911ENC_Inputs_Channel_2AT %I*ENC_Inputs_Channel_E5B5E92911ENC_Inputs_Channel_3AT %I*ENC_Inputs_Channel_E5B5E92911ENC_Inputs_Channel_4AT %I*ENC_Inputs_Channel_E5B5E92911PLS_InputsAT %I*PLS_Inputs_65C9A3D62DO_OutputsAT %Q*DO_Outputs_47E26D6A16AO_Outputs_Channel_1AT %Q*AO_Output_Channel_BA7EBB7C2AO_Outputs_Channel_2AT %Q*AO_Output_Channel_BA7EBB7C2AO_Outputs_Channel_3AT %Q*AO_Output_Channel_BA7EBB7C2AO_Outputs_Channel_4AT %Q*AO_Output_Channel_BA7EBB7C2ENC_Outputs_Channel_1AT %Q*ENC_Outputs_Channel_2E82BC435ENC_Outputs_Channel_2AT %Q*ENC_Outputs_Channel_2E82BC435ENC_Outputs_Channel_3AT %Q*ENC_Outputs_Channel_2E82BC435ENC_Outputs_Channel_4AT %Q*ENC_Outputs_Channel_2E82BC435PLS_OutputsAT %Q*PLS_Outputs_8EABC2241WcStateAT %I*WcState_9091E0EB2InfoDataAT %I*InfoData_32EB74EA10"}
{attribute addProperty CRC "261575999"}
{attribute addProperty Size "119"}
TYPE EM7004_0F97553F EXTENDS EtcSlaveTerminalBase_947E5A46 :
STRUCT
	{attribute addProperty Name "DI_Inputs"}
	DI_Inputs : DI_Inputs_9882B618;
	{attribute addProperty Name "ENC_Inputs_Channel_1"}
	ENC_Inputs_Channel_1 : ENC_Inputs_Channel_E5B5E929;
	{attribute addProperty Name "ENC_Inputs_Channel_2"}
	ENC_Inputs_Channel_2 : ENC_Inputs_Channel_E5B5E929;
	{attribute addProperty Name "ENC_Inputs_Channel_3"}
	ENC_Inputs_Channel_3 : ENC_Inputs_Channel_E5B5E929;
	{attribute addProperty Name "ENC_Inputs_Channel_4"}
	ENC_Inputs_Channel_4 : ENC_Inputs_Channel_E5B5E929;
	{attribute addProperty Name "PLS_Inputs"}
	PLS_Inputs : PLS_Inputs_65C9A3D6;
	{attribute addProperty Name "DO_Outputs"}
	DO_Outputs : DO_Outputs_47E26D6A;
	{attribute addProperty Name "AO_Outputs_Channel_1"}
	AO_Outputs_Channel_1 : AO_Output_Channel_BA7EBB7C;
	{attribute addProperty Name "AO_Outputs_Channel_2"}
	AO_Outputs_Channel_2 : AO_Output_Channel_BA7EBB7C;
	{attribute addProperty Name "AO_Outputs_Channel_3"}
	AO_Outputs_Channel_3 : AO_Output_Channel_BA7EBB7C;
	{attribute addProperty Name "AO_Outputs_Channel_4"}
	AO_Outputs_Channel_4 : AO_Output_Channel_BA7EBB7C;
	{attribute addProperty Name "ENC_Outputs_Channel_1"}
	ENC_Outputs_Channel_1 : ENC_Outputs_Channel_2E82BC43;
	{attribute addProperty Name "ENC_Outputs_Channel_2"}
	ENC_Outputs_Channel_2 : ENC_Outputs_Channel_2E82BC43;
	{attribute addProperty Name "ENC_Outputs_Channel_3"}
	ENC_Outputs_Channel_3 : ENC_Outputs_Channel_2E82BC43;
	{attribute addProperty Name "ENC_Outputs_Channel_4"}
	ENC_Outputs_Channel_4 : ENC_Outputs_Channel_2E82BC43;
	{attribute addProperty Name "PLS_Outputs"}
	PLS_Outputs : PLS_Outputs_8EABC224;
	{attribute addProperty Name "WcState"}
	WcState : WcState_9091E0EB;
	{attribute addProperty Name "InfoData"}
	InfoData : InfoData_32EB74EA;
END_STRUCT
END_TYPE

// ---- DUTs/IO/Devices/SyncUnitTask_2D604ED5.TcDUT
{attribute 'GeneratedUsingTerminal: IODEVICETYPE_ETHERCATPROT'}
{attribute addProperty BoxType "IODEVICETYPE_ETHERCATPROT"}
{attribute addProperty Id "WcStateAT %I*WcState_0B2B16F91InfoDataAT %I*InfoData_2A97D6CF8"}
{attribute addProperty CRC "761286357"}
{attribute addProperty Size "9"}
TYPE SyncUnitTask_2D604ED5 :
STRUCT
	{attribute addProperty Name "WcState"}
	WcState : WcState_0B2B16F9;
	{attribute addProperty Name "InfoData"}
	InfoData : InfoData_2A97D6CF;
END_STRUCT
END_TYPE

// ---- DUTs/IO/Devices/SyncUnitTasks_6FEB8257.TcDUT
{attribute 'GeneratedUsingTerminal: '}
{attribute addProperty BoxType ""}
{attribute addProperty Id "unreferencedAT %I*SyncUnitTask_2D604ED59PlcTaskAT %I*SyncUnitTask_2D604ED59"}
{attribute addProperty CRC "1877705303"}
{attribute addProperty Size "18"}
TYPE SyncUnitTasks_6FEB8257 :
STRUCT
	{attribute addProperty Name "unreferenced"}
	unreferenced : SyncUnitTask_2D604ED5;
	{attribute addProperty Name "PlcTask"}
	PlcTask : SyncUnitTask_2D604ED5;
END_STRUCT
END_TYPE

// ---- DUTs/IO/Devices/SyncUnits_99E584AF.TcDUT
{attribute 'GeneratedUsingTerminal: '}
{attribute addProperty BoxType ""}
{attribute addProperty Id "_defaultAT %I*SyncUnitTasks_6FEB825718"}
{attribute addProperty CRC "2581955759"}
{attribute addProperty Size "18"}
TYPE SyncUnits_99E584AF :
STRUCT
	{attribute addProperty Name "_default"}
	_default : SyncUnitTasks_6FEB8257;
END_STRUCT
END_TYPE

// ---- DUTs/IO/Topology/Beckhoff_EM2xxxEK1122_B7C04D41.TcDUT
{attribute 'GeneratedUsingTerminal: EK1122-0000-0018'}
{attribute addProperty BoxType "EK1122-0000-0018"}
{attribute addProperty Id "Beckhoff_EM2xxxsub_EK1100EK1100_1FC0878B2"}
{attribute addProperty CRC "3082833217"}
{attribute addProperty Size "2"}
{attribute addProperty Name "Beckhoff EM2xxxEK1122"}
TYPE Beckhoff_EM2xxxEK1122_B7C04D41 EXTENDS EK1122_1FC0878B :
STRUCT
	{attribute addProperty Name "Beckhoff EM2xxxsub EK1100"}
	{attribute addProperty PreviousPort "Beckhoff EM2xxxEK1122 : D"}
	Beckhoff_EM2xxxsub_EK1100 : EK1100_1FC0878B;
END_STRUCT
END_TYPE

// ---- DUTs/IO/Topology/Beckhoff_EM2xxx_23EB33C6.TcDUT
{attribute 'GeneratedUsingTerminal: EK1100-0000-0018'}
{attribute addProperty BoxType "EK1100-0000-0018"}
{attribute addProperty Id "Beckhoff_EM2xxxEK1122Beckhoff_EM2xxxEK1122_B7C04D412A_0001_EM2042_0000_0016EM2042_2B6483BD19A_0002_EM2042_0000_0017EM2042_2B6483BD19"}
{attribute addProperty CRC "602616774"}
{attribute addProperty Size "40"}
{attribute addProperty Name "Beckhoff EM2xxx"}
TYPE Beckhoff_EM2xxx_23EB33C6 EXTENDS EK1100_1FC0878B :
STRUCT
	{attribute addProperty Name "Beckhoff EM2xxxEK1122"}
	{attribute addProperty PreviousPort "Beckhoff EM2xxx : B"}
	Beckhoff_EM2xxxEK1122 : Beckhoff_EM2xxxEK1122_B7C04D41;
	{attribute addProperty Name "A_0001(EM2042-0000-0016)"}
	{attribute addProperty PreviousPort "Beckhoff EM2xxxEK1122 : C"}
	A_0001_EM2042_0000_0016 : EM2042_2B6483BD;
	{attribute addProperty Name "A_0002(EM2042-0000-0017)"}
	{attribute addProperty PreviousPort "A_0001(EM2042-0000-0016) : B"}
	A_0002_EM2042_0000_0017 : EM2042_2B6483BD;
END_STRUCT
END_TYPE

// ---- DUTs/IO/Topology/Beckhoff_EM3xxxEK1122_FEF78CCD.TcDUT
{attribute 'GeneratedUsingTerminal: EK1122-0000-0018'}
{attribute addProperty BoxType "EK1122-0000-0018"}
{attribute addProperty Id "Beckhoff_EM3xxxsub_EK1100EK1100_1FC0878B2"}
{attribute addProperty CRC "4277636301"}
{attribute addProperty Size "2"}
{attribute addProperty Name "Beckhoff EM3xxxEK1122"}
TYPE Beckhoff_EM3xxxEK1122_FEF78CCD EXTENDS EK1122_1FC0878B :
STRUCT
	{attribute addProperty Name "Beckhoff EM3xxxsub EK1100"}
	{attribute addProperty PreviousPort "Beckhoff EM3xxxEK1122 : D"}
	Beckhoff_EM3xxxsub_EK1100 : EK1100_1FC0878B;
END_STRUCT
END_TYPE

// ---- DUTs/IO/Topology/Beckhoff_EM3xxx_ABA31799.TcDUT
{attribute 'GeneratedUsingTerminal: EK1100-0000-0018'}
{attribute addProperty BoxType "EK1100-0000-0018"}
{attribute addProperty Id "Beckhoff_EM3xxxEK1122Beckhoff_EM3xxxEK1122_FEF78CCD2A_0001_EM3701_0000_0016EM3701_AB0D469D20A_0002_EM3702_0000_0016EM3702_FDD84FD828A_0003_EM3712_0000_0016EM3712_FDD84FD828"}
{attribute addProperty CRC "2879592345"}
{attribute addProperty Size "78"}
{attribute addProperty Name "Beckhoff EM3xxx"}
TYPE Beckhoff_EM3xxx_ABA31799 EXTENDS EK1100_1FC0878B :
STRUCT
	{attribute addProperty Name "Beckhoff EM3xxxEK1122"}
	{attribute addProperty PreviousPort "Beckhoff EM3xxx : B"}
	Beckhoff_EM3xxxEK1122 : Beckhoff_EM3xxxEK1122_FEF78CCD;
	{attribute addProperty Name "A_0001(EM3701-0000-0016)"}
	{attribute addProperty PreviousPort "Beckhoff EM3xxxEK1122 : C"}
	A_0001_EM3701_0000_0016 : EM3701_AB0D469D;
	{attribute addProperty Name "A_0002(EM3702-0000-0016)"}
	{attribute addProperty PreviousPort "A_0001(EM3701-0000-0016) : B"}
	A_0002_EM3702_0000_0016 : EM3702_FDD84FD8;
	{attribute addProperty Name "A_0003(EM3712-0000-0016)"}
	{attribute addProperty PreviousPort "A_0002(EM3702-0000-0016) : B"}
	A_0003_EM3712_0000_0016 : EM3712_FDD84FD8;
END_STRUCT
END_TYPE

// ---- DUTs/IO/Topology/Beckhoff_EM7xxxEK1122_DEE9974A.TcDUT
{attribute 'GeneratedUsingTerminal: EK1122-0000-0018'}
{attribute addProperty BoxType "EK1122-0000-0018"}
{attribute addProperty Id "Beckhoff_EM7xxxsub_EK1100EK1100_1FC0878B2"}
{attribute addProperty CRC "3739850570"}
{attribute addProperty Size "2"}
{attribute addProperty Name "Beckhoff EM7xxxEK1122"}
TYPE Beckhoff_EM7xxxEK1122_DEE9974A EXTENDS EK1122_1FC0878B :
STRUCT
	{attribute addProperty Name "Beckhoff EM7xxxsub EK1100"}
	{attribute addProperty PreviousPort "Beckhoff EM7xxxEK1122 : D"}
	Beckhoff_EM7xxxsub_EK1100 : EK1100_1FC0878B;
END_STRUCT
END_TYPE

// ---- DUTs/IO/Topology/Beckhoff_EM7xxx_9745B8AE.TcDUT
{attribute 'GeneratedUsingTerminal: EK1100-0000-0018'}
{attribute addProperty BoxType "EK1100-0000-0018"}
{attribute addProperty Id "Beckhoff_EM7xxxEK1122Beckhoff_EM7xxxEK1122_DEE9974A2A_0001_EM7004_0000_9995EM7004_866015E192A_0002_EM7004_0000_9996EM7004_7586CC95115A_0003_EM7004_0000_9997EM7004_7586CC95115A_0004_EM7004_0000_0016EM7004_5FA1DD22119A_0005_EM7004_0000_0017EM7004_0F97553F119A_0006_EM7004_0000_0018EM7004_0F97553F119"}
{attribute addProperty CRC "2537928878"}
{attribute addProperty Size "681"}
{attribute addProperty Name "Beckhoff EM7xxx"}
TYPE Beckhoff_EM7xxx_9745B8AE EXTENDS EK1100_1FC0878B :
STRUCT
	{attribute addProperty Name "Beckhoff EM7xxxEK1122"}
	{attribute addProperty PreviousPort "Beckhoff EM7xxx : B"}
	Beckhoff_EM7xxxEK1122 : Beckhoff_EM7xxxEK1122_DEE9974A;
	{attribute addProperty Name "A_0001(EM7004-0000-9995)"}
	{attribute addProperty PreviousPort "Beckhoff EM7xxxEK1122 : C"}
	A_0001_EM7004_0000_9995 : EM7004_866015E1;
	{attribute addProperty Name "A_0002(EM7004-0000-9996)"}
	{attribute addProperty PreviousPort "A_0001(EM7004-0000-9995) : B"}
	A_0002_EM7004_0000_9996 : EM7004_7586CC95;
	{attribute addProperty Name "A_0003(EM7004-0000-9997)"}
	{attribute addProperty PreviousPort "A_0002(EM7004-0000-9996) : B"}
	A_0003_EM7004_0000_9997 : EM7004_7586CC95;
	{attribute addProperty Name "A_0004(EM7004-0000-0016)"}
	{attribute addProperty PreviousPort "A_0003(EM7004-0000-9997) : B"}
	A_0004_EM7004_0000_0016 : EM7004_5FA1DD22;
	{attribute addProperty Name "A_0005(EM7004-0000-0017)"}
	{attribute addProperty PreviousPort "A_0004(EM7004-0000-0016) : B"}
	A_0005_EM7004_0000_0017 : EM7004_0F97553F;
	{attribute addProperty Name "A_0006(EM7004-0000-0018)"}
	{attribute addProperty PreviousPort "A_0005(EM7004-0000-0017) : B"}
	A_0006_EM7004_0000_0018 : EM7004_0F97553F;
END_STRUCT
END_TYPE

// ---- DUTs/IO/Topology/EtherCAT_Master_EMxxxx_E69B3047.TcDUT
{attribute 'GeneratedUsingTerminal: IODEVICETYPE_ETHERCATPROT'}
{attribute addProperty BoxType "IODEVICETYPE_ETHERCATPROT"}
{attribute addProperty Id "Beckhoff_EM2xxxBeckhoff_EM2xxx_23EB33C640Beckhoff_EM3xxxBeckhoff_EM3xxx_ABA3179978Beckhoff_EM7xxxBeckhoff_EM7xxx_9745B8AE681SyncUnitsSyncUnits_99E584AF18InputsInputs_25A0042B160OutputsOutputs_2397A10E106InfoDataInfoData_E68C61CD28"}
{attribute addProperty CRC "3868930119"}
{attribute addProperty Size "1111"}
{attribute addProperty Name "EtherCAT Master EMxxxx"}
TYPE EtherCAT_Master_EMxxxx_E69B3047 EXTENDS EtcMasterBase_62654B43 :
STRUCT
	{attribute addProperty Name "Beckhoff EM2xxx"}
	{attribute addProperty PreviousPort "EtherCAT Master EMxxxx : Master"}
	Beckhoff_EM2xxx : Beckhoff_EM2xxx_23EB33C6;
	{attribute addProperty Name "Beckhoff EM3xxx"}
	{attribute addProperty PreviousPort "Beckhoff EM2xxx : C"}
	Beckhoff_EM3xxx : Beckhoff_EM3xxx_ABA31799;
	{attribute addProperty Name "Beckhoff EM7xxx"}
	{attribute addProperty PreviousPort "Beckhoff EM3xxx : C"}
	Beckhoff_EM7xxx : Beckhoff_EM7xxx_9745B8AE;
	{attribute addProperty Name "SyncUnits"}
	SyncUnits : SyncUnits_99E584AF;
	{attribute addProperty Name "Inputs"}
	Inputs : Inputs_25A0042B;
	{attribute addProperty Name "Outputs"}
	Outputs : Outputs_2397A10E;
	{attribute addProperty Name "InfoData"}
	InfoData : InfoData_E68C61CD;
END_STRUCT
END_TYPE

// ---- DUTs/IO/Base/EtcSlaveBase_82538BE2.TcDUT

TYPE EtcSlaveBase_82538BE2 :
STRUCT
END_STRUCT
END_TYPE

// ---- DUTs/IO/Base/EtcSlaveBase_82538BE2.TcDUT

TYPE EtcSlaveBase_82538BE2 :
STRUCT
END_STRUCT
END_TYPE

// ---- DUTs/IO/Base/EtcSlaveBase_82538BE2.TcDUT

TYPE EtcSlaveBase_82538BE2 :
STRUCT
END_STRUCT
END_TYPE

// ---- DUTs/IO/Base/EtcSlaveTerminalBase_947E5A46.TcDUT

{attribute clr[Container(Layout.Stack)]}
{attribute clr[Group(Layout.GroupBox)]}
{attribute addProperty PreviousPort "Unknown"}
TYPE EtcSlaveTerminalBase_947E5A46 EXTENDS EtcSlaveBase_82538BE2 :
STRUCT
END_STRUCT
END_TYPE

// ---- DUTs/IO/Base/EtcSlaveBoxBase_77A0E4A7.TcDUT

{attribute clr[Container(Layout.Stack)]}
{attribute clr[Group(Layout.GroupBox)]}
{attribute addProperty PreviousPort "Unknown"}
TYPE EtcSlaveBoxBase_77A0E4A7 EXTENDS EtcSlaveBase_82538BE2 :
STRUCT
END_STRUCT
END_TYPE

// ---- DUTs/IO/Base/EtcSlaveEndTerminalBase_866C7F0C.TcDUT

{attribute clr[Container(Layout.Stack)]}
{attribute clr[Group(Layout.GroupBox)]}
{attribute addProperty PreviousPort "Unknown"}
TYPE EtcSlaveEndTerminalBase_866C7F0C EXTENDS EtcSlaveBase_82538BE2 :
STRUCT
END_STRUCT
END_TYPE

// ---- DUTs/IO/Base/InputBase_8311D824.TcDUT

TYPE InputBase_8311D824 :
STRUCT
END_STRUCT
END_TYPE

// ---- DUTs/IO/Base/OutputBase_10CEE7DE.TcDUT

TYPE OutputBase_10CEE7DE :
STRUCT
END_STRUCT
END_TYPE

// ---- DUTs/IO/Base/EtcMasterBase_62654B43.TcDUT

TYPE EtcMasterBase_62654B43 :
STRUCT
END_STRUCT
END_TYPE

// ---- GVLs/GVL_iXlinker.TcGVL
{attribute 'qualified_only'}
VAR_GLOBAL
		EtherCAT_Master_EMxxxx : EtherCAT_Master_EMxxxx_E69B3047;
END_VAR

// ---- POUs/MAIN.TcPOU
PROGRAM MAIN
VAR
END_VAR

END_PROGRAM
